    // IM5K4-PPM: 1 Axis
    {attribute 'pytmc' := 'pv: IM5K4:PPM:MMS'}
    {attribute 'TcLinkTo' := '.bLimitForwardEnable  := TIIB[IM5K4-EL7041-E1]^STM Status^Status^Digital input 1;
                              .bLimitBackwardEnable := TIIB[IM5K4-EL7041-E1]^STM Status^Status^Digital input 2;
                              .bBrakeRelease        := TIIB[IM5K4-EL2004-E3]^Channel 1^Output;
                              .nRawEncoderULINT     := TIIB[IM5K4-EL5042-E2]^FB Inputs Channel 1^Position'}
    M17: ST_MotionStage := (sName := 'IM5K4:PPM:MMS');

    // PF1K4-WFS_TARGET: 2 Axes
    {attribute 'pytmc' := 'pv: PF1K4:WFS:MMS:Y'}
    {attribute 'TcLinkTo' := '.bLimitForwardEnable  := TIIB[PF1K4-EL7041-E1]^STM Status^Status^Digital input 1;
                              .bLimitBackwardEnable := TIIB[PF1K4-EL7041-E1]^STM Status^Status^Digital input 2;
                              .bBrakeRelease        := TIIB[PF1K4-EL2004-E4]^Channel 1^Output;
                              .nRawEncoderULINT     := TIIB[PF1K4-EL5042-E3]^FB Inputs Channel 2^Position'}
    M18: ST_MotionStage := (sName := 'PF1K4:WFS:MMS:Y');
    {attribute 'pytmc' := 'pv: PF1K4:WFS:MMS:Z'}
    {attribute 'TcLinkTo' := '.nRawEncoderULINT     := TIIB[PF1K4-EL5042-E3]^FB Inputs Channel 1^Position'}
    M19: ST_MotionStage := (sName := 'PF1K4:WFS:MMS:Z');

    // LI1K4-IP1: 1 Axis
    {attribute 'pytmc' := 'pv: LI1K4:IP1:MMS'}
    {attribute 'TcLinkTo' := '.bLimitForwardEnable  := TIIB[LI1K4-EL7041-E1]^STM Status^Status^Digital input 1;
                              .bLimitBackwardEnable := TIIB[LI1K4-EL7041-E1]^STM Status^Status^Digital input 2;
                              .bBrakeRelease        := TIIB[LI1K4-EL2004-E3]^Channel 1^Output;
                              .nRawEncoderULINT     := TIIB[LI1K4-EL5042-E2]^FB Inputs Channel 1^Position'}
    M20: ST_MotionStage := (sName := 'LI1K4:IP1:MMS');

    // TM1K4: 2 Axes
    {attribute 'pytmc' := 'pv: TM1K4:ATM:MMS:Y'}
    {attribute 'TcLinkTo' := '.bLimitForwardEnable  := TIIB[TM1K4-EL7041-E1]^STM Status^Status^Digital input 1;
                              .bLimitBackwardEnable := TIIB[TM1K4-EL7041-E1]^STM Status^Status^Digital input 2;
                              .bBrakeRelease        := TIIB[TM1K4-EL2004-E4]^Channel 1^Output;
                              .nRawEncoderULINT     := TIIB[TM1K4-EL5042-E3]^FB Inputs Channel 1^Position'}
    M21: ST_MotionStage := (sName := 'TM1K4:ATM:MMS:Y');
    {attribute 'pytmc' := 'pv: TM1K4:ATM:MMS:X'}
    {attribute 'TcLinkTo' := '.nRawEncoderULINT     := TIIB[TM1K4-EL5042-E3]^FB Inputs Channel 2^Position'}
    M22: ST_MotionStage := (sName := 'TM1K4:ATM:MMS:X');

  (*   // SL2K4-SCATTER: 4 Axes
    {attribute 'pytmc' := 'pv: SL2K4:SCATTER:MMS:BOTTOM'}
    {attribute 'TcLinkTo' := '.bLimitForwardEnable  := TIIB[SL2K4-EL7031-E1]^STM Status^Status^Digital input 2;
                             .bLimitBackwardEnable := TIIB[SL2K4-EL7031-E1]^STM Status^Status^Digital input 1;
                              .nRawEncoderUINT      := TIIB[SL2K4-EL5101-E2]^ENC Status compact^Counter value'}
    M23: ST_MotionStage := (sName := 'SL2K4:SCATTER:MMS:BOTTOM');
    {attribute 'pytmc' := 'pv: SL2K4:SCATTER:MMS:TOP'}
    {attribute 'TcLinkTo' := '.bLimitForwardEnable  := TIIB[SL2K4-EL7031-E3]^STM Status^Status^Digital input 2;
                              .bLimitBackwardEnable := TIIB[SL2K4-EL7031-E3]^STM Status^Status^Digital input 1;
                              .nRawEncoderUINT      := TIIB[SL2K4-EL5101-E4]^ENC Status compact^Counter value'}
    M24: ST_MotionStage := (sName := 'SL2K4:SCATTER:MMS:TOP');
    {attribute 'pytmc' := 'pv: SL2K4:SCATTER:MMS:NORTH'}
    {attribute 'TcLinkTo' := '.bLimitForwardEnable  := TIIB[SL2K4-EL7031-E5]^STM Status^Status^Digital input 1;
                              .bLimitBackwardEnable := TIIB[SL2K4-EL7031-E5]^STM Status^Status^Digital input 2;
                              .nRawEncoderUINT      := TIIB[SL2K4-EL5101-E6]^ENC Status compact^Counter value'}
    M25: ST_MotionStage := (sName := 'SL2K4:SCATTER:MMS:NORTH');
    {attribute 'pytmc' := 'pv: SL2K4:SCATTER:MMS:SOUTH'}
    {attribute 'TcLinkTo' := '.bLimitForwardEnable  := TIIB[SL2K4-EL7031-E7]^STM Status^Status^Digital input 1;
                              .bLimitBackwardEnable := TIIB[SL2K4-EL7031-E7]^STM Status^Status^Digital input 2;
                              .nRawEncoderUINT      := TIIB[SL2K4-EL5101-E8]^ENC Status compact^Counter value'}
    M26: ST_MotionStage := (sName := 'SL2K4:SCATTER:MMS:SOUTH');
    *)

    // IM6K4-PPM: 1 Axis
    {attribute 'pytmc' := 'pv: IM6K4:PPM:MMS'}
    {attribute 'TcLinkTo' := '.bLimitForwardEnable  := TIIB[IM6K4-EL7041-E1]^STM Status^Status^Digital input 1;
                              .bLimitBackwardEnable := TIIB[IM6K4-EL7041-E1]^STM Status^Status^Digital input 2;
                              .bBrakeRelease        := TIIB[IM6K4-EL2004-E3]^Channel 1^Output;
                              .nRawEncoderULINT     := TIIB[IM6K4-EL5042-E2]^FB Inputs Channel 1^Position'}
    M27: ST_MotionStage := (sName := 'IM6K4:PPM:MMS');

    // PF2K4-WFS_TARGET: 2 Axes
    {attribute 'pytmc' := 'pv: PF2K4:WFS:MMS:Y'}
    {attribute 'TcLinkTo' := '.bLimitForwardEnable  := TIIB[PF2K4-EL7041-E1]^STM Status^Status^Digital input 1;
                              .bLimitBackwardEnable := TIIB[PF2K4-EL7041-E1]^STM Status^Status^Digital input 2;
                              .bBrakeRelease        := TIIB[PF2K4-EL2004-E4]^Channel 1^Output;
                              .nRawEncoderULINT     := TIIB[PF2K4-EL5042-E3]^FB Inputs Channel 2^Position'}
    M28: ST_MotionStage := (sName := 'PF2K4:WFS:MMS:Y');
    {attribute 'pytmc' := 'pv: PF2K4:WFS:MMS:Z'}
    {attribute 'TcLinkTo' := '.nRawEncoderULINT     := TIIB[PF2K4-EL5042-E3]^FB Inputs Channel 1^Position'}
    M29: ST_MotionStage := (sName := 'PF2K4:WFS:MMS:Z');

    // TM2K4 2 Axes
    {attribute 'pytmc' := 'pv: TM2K4:ATM:MMS:Y'}
    {attribute 'TcLinkTo' := '.bLimitForwardEnable  := TIIB[TM2K4-EL7041-E1]^STM Status^Status^Digital input 1;
                              .bLimitBackwardEnable := TIIB[TM2K4-EL7041-E1]^STM Status^Status^Digital input 2;
                              .bBrakeRelease        := TIIB[TM2K4-EL2004-E4]^Channel 1^Output;
                              .nRawEncoderULINT     := TIIB[TM2K4-EL5042-E3]^FB Inputs Channel 1^Position'}
    M30: ST_MotionStage := (sName := 'TM2K4:ATM:MMS:Y');
    {attribute 'pytmc' := 'pv: TM2K4:ATM:MMS:X'}
    {attribute 'TcLinkTo' := '.nRawEncoderULINT     := TIIB[TM2K4-EL5042-E3]^FB Inputs Channel 2^Position'}
    M31: ST_MotionStage := (sName := 'TM2K4:ATM:MMS:X');

    // SP1K4 14 Axes
    {attribute 'pytmc' := '
        pv: TMO:SPEC:MMS:01
    '}
    // Lens X (not use it after July 2023)
    M32 : ST_MotionStage := (
        bHardwareEnable:=TRUE,
        bPowerSelf:=TRUE,
        nEnableMode:=ENUM_StageEnableMode.DURING_MOTION,
        nHomingMode := ENUM_EpicsHomeCmd.ABSOLUTE_SET);
    {attribute 'TcLinkTo' := '.bLimitForwardEnable:=TIIB[FoilX-EL7041]^STM Status^Status^Digital input 2;
                              .bLimitBackwardEnable:=TIIB[FoilX-EL7041]^STM Status^Status^Digital input 1'
                              .nRawEncoderULINT:=TIIB[SP1K4-EL5042-E2]^FB Inputs Channel 2^Position'}
    {attribute 'pytmc' := '
        pv: TMO:SPEC:MMS:02
    '}
    // solid atten X(Foil X)
    M33: ST_MotionStage := (
        bHardwareEnable:=TRUE,
        bPowerSelf:=FALSE,
        nEnableMode:=ENUM_StageEnableMode.DURING_MOTION,
        nHomingMode := ENUM_EpicsHomeCmd.NONE,
        sName := 'TMO:SPEC:MMS:02');
    {attribute 'TcLinkTo' := '.bLimitForwardEnable:=TIIB[ZonePlateX-EL7041]^STM Status^Status^Digital input 2;
                              .bLimitBackwardEnable:=TIIB[ZonePlateX-EL7041]^STM Status^Status^Digital input 1'
                              .nRawEncoderULINT:=TIIB[SP1K4-EL5042-E1]^FB Inputs Channel 1^Position'}
    {attribute 'pytmc' := '
        pv: TMO:SPEC:MMS:03
    '}
    // Zone Plate X
    M34 : ST_MotionStage := (
        bHardwareEnable:=TRUE,
        bPowerSelf:=FALSE,
        nEnableMode:=ENUM_StageEnableMode.DURING_MOTION,
        sName := 'TMO:SPEC:MMS:03');
    {attribute 'TcLinkTo' := '.bLimitForwardEnable:=TIIB[ZonePlateY-EL7041]^STM Status^Status^Digital input 2;
                              .bLimitBackwardEnable:=TIIB[ZonePlateY-EL7041]^STM Status^Status^Digital input 1';
                              .nRawEncoderULINT:=TIIB[SP1K4-EL5042-E1]^FB Inputs Channel 2^Position'}
    {attribute 'pytmc' := '
        pv: TMO:SPEC:MMS:04
    '}
    // Zone Plate Y
    M35 : ST_MotionStage := (
        bHardwareEnable:=TRUE,
        bPowerSelf:=FALSE,
        nEnableMode:=ENUM_StageEnableMode.DURING_MOTION,
        sName := 'TMO:SPEC:MMS:04');
    {attribute 'TcLinkTo' := '.bLimitForwardEnable:=TIIB[ZonePlateZ-EL7041]^STM Status^Status^Digital input 1;
                              .bLimitBackwardEnable:=TIIB[ZonePlateZ-EL7041]^STM Status^Status^Digital input 2';
                              .nRawEncoderULINT:=TIIB[SP1K4-EL5042-E2]^FB Inputs Channel 1^Position'}
    {attribute 'pytmc' := '
        pv: TMO:SPEC:MMS:05
    '}
    // Zone Plate Z
    M36 : ST_MotionStage := (
        bHardwareEnable:=TRUE,
        bPowerSelf:=FALSE,
        nEnableMode:=ENUM_StageEnableMode.DURING_MOTION,
        sName := 'TMO:SPEC:MMS:05');
    {attribute 'TcLinkTo' := '.bLimitForwardEnable:=TIIB[YagX-EL7041]^STM Status^Status^Digital input 2;
                              .bLimitBackwardEnable:=TIIB[YagX-EL7041]^STM Status^Status^Digital input 1';
                              .nRawEncoderULINT:=TIIB[SP1K4-EL5042-E8]^FB Inputs Channel 1^Position'}

    {attribute 'pytmc' := '
        pv: TMO:SPEC:MMS:06
    '}
    // Yag X
    M37 : ST_MotionStage := (
        bHardwareEnable:=TRUE,
        bPowerSelf:=TRUE,
        nEnableMode:=ENUM_StageEnableMode.DURING_MOTION,
        nHomingMode := ENUM_EpicsHomeCmd.ABSOLUTE_SET);
    {attribute 'TcLinkTo' := '.bLimitForwardEnable:=TIIB[YagY-EL7041]^STM Status^Status^Digital input 1;
                              .bLimitBackwardEnable:=TIIB[YagY-EL7041]^STM Status^Status^Digital input 2'}

    {attribute 'pytmc' := '
        pv: TMO:SPEC:MMS:07
    '}
    // Yag Y
    M38 : ST_MotionStage := (
        bHardwareEnable:=TRUE,
        bPowerSelf:=TRUE,
        nEnableMode:=ENUM_StageEnableMode.DURING_MOTION,
        nHomingMode := ENUM_EpicsHomeCmd.ABSOLUTE_SET);

    {attribute 'TcLinkTo' := '.bLimitForwardEnable:=TIIB[YagZ-EL7041]^STM Status^Status^Digital input 2;
                              .bLimitBackwardEnable:=TIIB[YagZ-EL7041]^STM Status^Status^Digital input 1';
                              .nRawEncoderULINT:=TIIB[SP1K4-EL5042-E8]^FB Inputs Channel 2^Position'}

    {attribute 'pytmc' := '
        pv: TMO:SPEC:MMS:08
    '}
    // Yag Z
    M39 : ST_MotionStage := (
        bHardwareEnable:=TRUE,
        bPowerSelf:=TRUE,
        nEnableMode:=ENUM_StageEnableMode.DURING_MOTION,
        nHomingMode := ENUM_EpicsHomeCmd.ABSOLUTE_SET);
    {attribute 'TcLinkTo' := '.bLimitForwardEnable:=TIIB[YagTheta-EL7041]^STM Status^Status^Digital input 1;
                              .bLimitBackwardEnable:=TIIB[YagTheta-EL7041]^STM Status^Status^Digital input 2'}
    {attribute 'pytmc' := '
        pv: TMO:SPEC:MMS:09
    '}
    // Yag Theta
    M40 : ST_MotionStage := (
        bHardwareEnable:=TRUE,
        bPowerSelf:=TRUE,
        nEnableMode:=ENUM_StageEnableMode.DURING_MOTION,
        nHomingMode := ENUM_EpicsHomeCmd.ABSOLUTE_SET);
    {attribute 'pytmc' := '
        pv: TMO:SPEC:MMS:10
    '}
    // Thorlabs1
    M41 : ST_MotionStage := (
        bHardwareEnable:=TRUE,
        bPowerSelf:=TRUE,
        nEnableMode:=ENUM_StageEnableMode.DURING_MOTION,
        nHomingMode := ENUM_EpicsHomeCmd.ABSOLUTE_SET);
    {attribute 'pytmc' := '
        pv: TMO:SPEC:MMS:11
    '}
    // Thorlabs2
    M42 : ST_MotionStage := (
        bHardwareEnable:=TRUE,
        bPowerSelf:=TRUE,
        nEnableMode:=ENUM_StageEnableMode.DURING_MOTION,
        nHomingMode := ENUM_EpicsHomeCmd.ABSOLUTE_SET);

    {attribute 'pytmc' := '
        pv: TMO:SPEC:MMS:12
    '}
    //thorlab-lenX
    M43 : ST_MotionStage := (
        bHardwareEnable:=TRUE,
        bPowerSelf:=TRUE,
        nEnableMode:=ENUM_StageEnableMode.DURING_MOTION,
        nHomingMode := ENUM_EpicsHomeCmd.ABSOLUTE_SET);

    {attribute 'TcLinkTo' := '.bLimitForwardEnable:=TIIB[FoilY-EL7041]^STM Status^Status^Digital input 1;
                              .bLimitBackwardEnable:=TIIB[FoilY-EL7041]^STM Status^Status^Digital input 2';
                               .nRawEncoderULINT:=TIIB[SP1K4-EL5042-E7]^FB Inputs Channel 2^Position'}
    {attribute 'pytmc' := '
        pv: TMO:SPEC:MMS:13
    '}
     //Solid att Y(FOIL-Y)
    M44 : ST_MotionStage := (
        bHardwareEnable:=TRUE,
        bPowerSelf:=FALSE,
        nEnableMode:=ENUM_StageEnableMode.DURING_MOTION,
        nHomingMode := ENUM_EpicsHomeCmd.NONE,
        sName := 'TMO:SPEC:MMS:13');

 // LI2K4-MMS: Y

    {attribute 'TcLinkTo' := '.bLimitForwardEnable  := TIIB[LI2K4Y-EL7047-E1]^STM Status^Status^Digital input 1;
                              .bLimitBackwardEnable := TIIB[LI2K4Y-EL7047-E1]^STM Status^Status^Digital input 2;
                              .nRawEncoderULINT     := TIIB[LI2K4-EL5042-E2]^FB Inputs Channel 1^Position'}
    {attribute 'pytmc' := '
        pv: LI2K4:IP1:MMS:Y
    '}

    M45: ST_MotionStage := (
        bHardwareEnable:=TRUE,
        bPowerSelf:=FALSE,
        nEnableMode:=ENUM_StageEnableMode.DURING_MOTION,
        nHomingMode := ENUM_EpicsHomeCmd.NONE,
        sName := 'LI2K4:IP1:MMS:Y');
// LI2K4-MMS: X
    {attribute 'TcLinkTo' := '.bLimitForwardEnable  := TIIB[LI2K4X-EL7047-E3]^STM Status^Status^Digital input 1;
                              .bLimitBackwardEnable := TIIB[LI2K4X-EL7047-E3]^STM Status^Status^Digital input 2;
                              .nRawEncoderULINT     := TIIB[LI2K4-EL5042-E2]^FB Inputs Channel 2^Position'}
    {attribute 'pytmc' := '
        pv: LI2K4:IP1:MMS:X
    '}
    M46: ST_MotionStage := (
        bHardwareEnable:=TRUE,
        bPowerSelf:=FALSE,
        nEnableMode:=ENUM_StageEnableMode.DURING_MOTION,
        nHomingMode := ENUM_EpicsHomeCmd.NONE,
        sName := 'LI2K4:IP1:MMS:X');

    //PA1K4-PF-MMS-Y
     {attribute 'TcLinkTo' := '.bLimitForwardEnable  := TIIB[PA1K4-PF-EL7047-E4]^STM Status^Status^Digital input 1;
                              .bLimitBackwardEnable := TIIB[PA1K4-PF-EL7047-E4]^STM Status^Status^Digital input 2;
                              .nRawEncoderULINT     := TIIB[PA1K4-PF-EL5042-E5]^FB Inputs Channel 1^Position'}
    {attribute 'pytmc' := '
        pv: PA1K4:PF:MMS:Y
    '}
    M47: ST_MotionStage := (
        bHardwareEnable:=TRUE,
        bPowerSelf:=FALSE,
        nEnableMode:=ENUM_StageEnableMode.DURING_MOTION,
        nHomingMode := ENUM_EpicsHomeCmd.NONE,
        sName := 'PA1K4:PF:MMS:Y');

END_VAR

// ---- POUs/FB_SP_ZP.TcPOU
FUNCTION_BLOCK FB_SP_ZP
VAR_IN_out
     stXStage: ST_MotionStage;
     stYStage: ST_MotionStage;
     stZStage: ST_MotionStage;
    fbArbiter: FB_Arbiter;
    fbFFHWO: FB_HardwareFFOutput;
END_VAR
VAR_INPUT
    stOut: DUT_PositionState;
    stYag: DUT_PositionState;
    stNe1: DUT_PositionState;
    stNe2: DUT_PositionState;
    stNe3: DUT_PositionState;
    st3w1: DUT_PositionState;
    st3w2: DUT_PositionState;
    stO2: DUT_PositionState;
    stO1: DUT_PositionState;
    stTi1: DUT_PositionState;
    stTi2: DUT_PositionState;
    stN1: DUT_PositionState;
    stN2:DUT_PositionState;
    stC1: DUT_PositionState;
    stC2: DUT_PositionState;
    //nTransitionAssertionID: UDINT;
    //nUnknownAssertionID: UDINT;

          {attribute 'pytmc' := '
        pv: MMS:X:STATE
        io: i
    '}
    fbStates_x: FB_ZonePlate_States;

       {attribute 'pytmc' := '
        pv: MMS:Y:STATE
        io: i
    '}
    fbStates_y: FB_ZonePlate_States;

    zp_enumSet : ENUM_ZonePlate_States;
END_VAR
VAR
     fbXStage: FB_MotionStage;
     fbYStage: FB_MotionStage;
     fbZStage: FB_MotionStage;

    (*FFO*)

    FFO: FB_fastFault :=(
        i_DevName:= 'SP1K4',
        i_Desc := 'Fault Occures when the X and Y states d not match',
        i_TypeCode := 16#300 //todo find a type code on confluence
        );


END_VAR

fbXStage(stMotionStage:=stXStage);
stXStage.bHardwareEnable := TRUE;
stXStage.bPowerSelf := FALSE;
stXStage.nEnableMode := ENUM_StageEnableMode.DURING_MOTION;

fbYStage(stMotionStage:=stYStage);
stYStage.bHardwareEnable := TRUE;
stYStage.bPowerSelf := FALSE;
stYStage.nEnableMode := ENUM_StageEnableMode.DURING_MOTION;

fbZStage(stMotionStage:=stZStage);
stZStage.bHardwareEnable := TRUE;
stZStage.bPowerSelf := FALSE;
stZStage.nEnableMode := ENUM_StageEnableMode.DURING_MOTION;





//TODO write the Y and X position before calling the function

fbStates_X(
    fbArbiter:=fbArbiter,
    fbFFHWO:=fbFFHWO,
 //   nTransitionAssertionID:=nTransitionAssertionID,
 //   nUnknownAssertionID:=nUnknownAssertionID,
    stMotionStage:=stXStage,
    bEnable:=TRUE,
    enumSet:= zp_enumSet,
    stOut:=stOut,
    stYag :=stYag,
    stNe1:=stNe1,
    stNe2:=stNe2,
    stNe3:=stNe3,
    st3w1:=st3w1,
    st3w2:=st3w2,
    stO2:=stO2,
    stO1:=stO1,
    stTi1:=stTi1,
    stTi2:=stTi2,
    stN1:=stN1,
    stN2:=stN2,
    stC1:=stC1,
    stC2:=stC2,
  ); //TODO ADD all other states




fbStates_Y(
    fbArbiter:=fbArbiter,
    fbFFHWO:=fbFFHWO,
 //   nTransitionAssertionID:=nTransitionAssertionID,
//    nUnknownAssertionID:=nUnknownAssertionID,
    stMotionStage:=stYStage,
    bEnable:=TRUE,
    enumSet:= zp_enumSet,
    stOut:=stOut,
    stYag:=stYag,
    stNe1:=stNe1,
    stNe2:=stNe2,
    stNe3:=stNe3,
    st3w1:=st3w1,
    st3w2:=st3w2,
    stO2:=stO2,
    stO1:=stO1,
    stTi1:=stTi1,
    stTi2:=stTi2,
    stN1:=stN1,
    stN2:=stN2,
    stC1:=stC1,
    stC2:=stC2,
);


    FFO(i_xOK:= (fbStates_X.enumGet = fbStates_Y.enumGet),
    io_fbFFHWO:= fbFFHWO,
    i_xAutoReset := TRUE );

END_FUNCTION_BLOCK

// ---- POUs/temp/FB_ZonePlate_States.TcPOU
FUNCTION_BLOCK FB_ZonePlate_States EXTENDS FB_PositionStateBase_WithPMPS
VAR_INPUT
     {attribute 'pytmc' := '
        pv: SET
        io: io
    '}
    enumSet: ENUM_ZonePlate_States;
    stOut: DUT_PositionState;
    stYag: DUT_PositionState;
    stNe1: DUT_PositionState;
    stNe2: DUT_PositionState;
    stNe3: DUT_PositionState;
    st3w1: DUT_PositionState;
    st3w2: DUT_PositionState;
    stO1: DUT_PositionState;
    stO2: DUT_PositionState;
    stTi1: DUT_PositionState;
    stTi2: DUT_PositionState;
    stN1: DUT_PositionState;
    stN2:DUT_PositionState;
    stC1: DUT_PositionState;
    stC2: DUT_PositionState;
    stW1: DuT_PositionState;
END_VAR
VAR_OUTPUT
     {attribute 'pytmc' := '
        pv: GET
        io: i
    '}
    enumGet: ENUM_ZonePlate_States;
END_VAR
VAR
    bInittwo: BOOL := TRUE;
    fbStateDefaults: FB_PositionState_Defaults;
    // These are the default values
    // Set values on states prior to passing in for non-default values
    //TODO correct these default positions
    fDelta: LREAL := 1;
    fVelocity: LREAL := 5;
    fAccel: LREAL := 200;
    fDecel: LREAL := 25;
END_VAR

//State init
IF (bInittwo) THEN
    bInittwo := FALSE;
    //Set theses for every state
    stOut.sName := 'OUT';
    stOut.bUseRawCounts:= FALSE;
    stOut.bValid := TRUE;
        fbStateDefaults(
        stPositionState:=stOut,
        fVeloDefault:=fVelocity,
        fDeltaDefault:=fDelta,
        fAccelDefault:=fAccel,
        fDecelDefault:=fDecel,
    );
    stYag.sName := 'Yag';
    stYag.bUseRawCounts:= FALSE;
    stYag.bValid := TRUE;
        fbStateDefaults(
        stPositionState:=stYag,
        fVeloDefault:=fVelocity,
        fDeltaDefault:=fDelta,
        fAccelDefault:=fAccel,
        fDecelDefault:=fDecel,
    );
    stNe1.sName := 'Ne1';
    stNe1.bUseRawCounts:= FALSE;
    stNe1.bValid := TRUE;
        fbStateDefaults(
        stPositionState:=stNe1,
        fVeloDefault:=fVelocity,
        fDeltaDefault:=fDelta,
        fAccelDefault:=fAccel,
        fDecelDefault:=fDecel,
    );
    stNe2.sName := 'Ne2';
    stNe2.bUseRawCounts:= FALSE;
    stNe2.bValid := TRUE;
        fbStateDefaults(
        stPositionState:=stNe2,
        fVeloDefault:=fVelocity,
        fDeltaDefault:=fDelta,
        fAccelDefault:=fAccel,
        fDecelDefault:=fDecel,
    );
    stNe3.sName := 'Ne3';
    stNe3.bUseRawCounts:= FALSE;
    stNe3.bValid := TRUE;
        fbStateDefaults(
        stPositionState:=stNe3,
        fVeloDefault:=fVelocity,
        fDeltaDefault:=fDelta,
        fAccelDefault:=fAccel,
        fDecelDefault:=fDecel,
    );
    st3w1.sName := '3w1';
    st3w1.bUseRawCounts:= FALSE;
    st3w1.bValid := TRUE;
        fbStateDefaults(
        stPositionState:=st3w1,
        fVeloDefault:=fVelocity,
        fDeltaDefault:=fDelta,
        fAccelDefault:=fAccel,
        fDecelDefault:=fDecel,
    );
    st3w2.sName := '3w2';
    st3w2.bUseRawCounts:= FALSE;
    st3w2.bValid := TRUE;
        fbStateDefaults(
        stPositionState:=st3w2,
        fVeloDefault:=fVelocity,
        fDeltaDefault:=fDelta,
        fAccelDefault:=fAccel,
        fDecelDefault:=fDecel,
    );
    stO1.sName := 'O1';
    stO1.bUseRawCounts:= FALSE;
    stO1.bValid := TRUE;
        fbStateDefaults(
        stPositionState:=stO1,
        fVeloDefault:=fVelocity,
        fDeltaDefault:=fDelta,
        fAccelDefault:=fAccel,
        fDecelDefault:=fDecel,
    );
    stO2.sName := 'O2';
    stO2.bUseRawCounts:= FALSE;
    stO2.bValid := TRUE;
        fbStateDefaults(
        stPositionState:=stO2,
        fVeloDefault:=fVelocity,
        fDeltaDefault:=fDelta,
        fAccelDefault:=fAccel,
        fDecelDefault:=fDecel,
    );

    stTi1.sName := 'Ti1';
    stTi1.bUseRawCounts:= FALSE;
    stTi1.bValid := TRUE;
        fbStateDefaults(
        stPositionState:=stTi1,
        fVeloDefault:=fVelocity,
        fDeltaDefault:=fDelta,
        fAccelDefault:=fAccel,
        fDecelDefault:=fDecel,
    );
    stTi2.sName := 'Ti2';
    stTi2.bUseRawCounts:= FALSE;
    stTi2.bValid := TRUE;
        fbStateDefaults(
        stPositionState:=stTi2,
        fVeloDefault:=fVelocity,
        fDeltaDefault:=fDelta,
        fAccelDefault:=fAccel,
        fDecelDefault:=fDecel,
    );
    stN1.sName := 'N1';
    stN1.bUseRawCounts:= FALSE;
    stN1.bValid := TRUE;
        fbStateDefaults(
        stPositionState:=stN1,
        fVeloDefault:=fVelocity,
        fDeltaDefault:=fDelta,
        fAccelDefault:=fAccel,
        fDecelDefault:=fDecel,
    );
    stN2.sName := 'N2';
    stN2.bUseRawCounts:= FALSE;
    stN2.bValid := TRUE;
        fbStateDefaults(
        stPositionState:=stN2,
        fVeloDefault:=fVelocity,
        fDeltaDefault:=fDelta,
        fAccelDefault:=fAccel,
        fDecelDefault:=fDecel,
    );
    stC1.sName := 'C1';
    stC1.bUseRawCounts:= FALSE;
    stC1.bValid := TRUE;
        fbStateDefaults(
        stPositionState:=stC1,
        fVeloDefault:=fVelocity,
        fDeltaDefault:=fDelta,
        fAccelDefault:=fAccel,
        fDecelDefault:=fDecel,
    );
    stC2.sName := 'C2';
    stC2.bUseRawCounts:= FALSE;
    stC2.bValid := TRUE;
        fbStateDefaults(
        stPositionState:=stC2,
        fVeloDefault:=fVelocity,
        fDeltaDefault:=fDelta,
        fAccelDefault:=fAccel,
        fDecelDefault:=fDecel,
    );
    stW1.sName := 'W1';
    stW1.bUseRawCounts:= FALSE;
    stW1.bValid := TRUE;
        fbStateDefaults(
        stPositionState:=stW1,
        fVeloDefault:=fVelocity,
        fDeltaDefault:=fDelta,
        fAccelDefault:=fAccel,
        fDecelDefault:=fDecel,
    );

//Add all states

    arrStates[1] := stOut;
    arrStates[2] := stYag;
    arrStates[3] := stNe1;
    arrStates[4] := stNe2;
    arrStates[5] := stNe3;
    arrStates[6] := st3w1;
    arrStates[7] := st3w2;
    arrStates[8] := stO1;
    arrStates[9] := stO2;
    arrStates[10] := stTi1;
    arrStates[11] := stTi2;
    arrStates[12] := stN1;
    arrStates[13] := stN2;
    arrStates[14] := stC1;
    arrStates[15] := stC2;
 //   arrStates[16] := stW1;

END_IF

setState := enumSet;
Exec();
enumGet := getState;
enumSet := setState;

END_FUNCTION_BLOCK

// ---- POUs/PRG_1_PlcTask.TcPOU
PROGRAM PRG_1_PlcTask
VAR
END_VAR

PRG_2_PMPS_PRE();

PRG_AL1K4_L2SI();
PRG_IM2K4_PPM();
PRG_IM3K4_PPM();
PRG_IM4K4_PPM();
PRG_IM5K4_PPM();
PRG_IM6K4_PPM();
PRG_LI1K4_IP1();
PRG_PF1K4_WFS_TARGET();
PRG_PF2K4_WFS_TARGET();
PRG_SL1K4_SCATTER();
//PRG_SL2K4_SCATTER();
PRG_ST4K4_TMO_TERM();
PRG_PC5K4();
//PRG_ST5K4_TMO_TERM_FIXED();
PRG_TM1K4();
PRG_TM2K4();
PRG_SP1K4();
PRG_LI2K4_IP1();
PRG_PA1K4_PF();


PRG_3_PMPS_POST();
PRG_4_LOG();

END_PROGRAM

// ---- POUs/PRG_2_PMPS_PRE.TcPOU
PROGRAM PRG_2_PMPS_PRE
VAR
END_VAR

MOTION_GVL.fbStandardPMPSDB(
    io_fbFFHWO:=GVL_PMPS.fbFastFaultOutput1,
    bEnable:=TRUE,
    sPLCName:='plc-tmo-motion',
    sDirectory:='/home/ecs-user/pmpsdb/'
    );

END_PROGRAM

// ---- POUs/PRG_AL1K4_L2SI.TcPOU
PROGRAM PRG_AL1K4_L2SI
VAR
    {attribute 'pytmc' := '
        pv: AL1K4:L2SI
        io: io
    '}
    {attribute 'TcLinkTo' := '.fbLaser.iLaserINT := TIIB[AL1K4-EL4004-E4]^AO Outputs Channel 1^Analog output;
                              .fbLaser.iShutdownINT := TIIB[AL1K4-EL4004-E4]^AO Outputs Channel 2^Analog output'}
    fbAL1K4: FB_REF;
    fbStateSetup: FB_StateSetupHelper;
    stDefault: ST_PositionState :=(
        fVelocity := 1,
        bMoveOK := TRUE,
        bValid := TRUE
    );
//    bInit: BOOL;
END_VAR


fbStateSetup(StPositionState:=stDefault, bSetDefault:=TRUE);
fbStateSetup(StPositionState:=fbAL1K4.stOut, fposition:=-33.5, sPmpsState := 'AL1K4:L2SI-OUT');
fbStateSetup(StPositionState:=fbAL1K4.stIn, fposition:=-75, sPmpsState := 'AL1K4:L2SI-IN');
{*
//fbAL1K4.stOut.fPosition := -33.5; // Upper limit
fbAL1K4.stOut.bUseRawCounts := FALSE;
fbAL1K4.stOut.bValid := TRUE;
fbAL1K4.stOut.bMoveOk := TRUE;
fbAL1K4.stOut.stPMPS.sPmpsState := 'AL1K4:L2SI-OUT';

//fbAL1K4.stIn.fPosition := -75; // Current position at time of edit
fbAL1K4.stIn.bUseRawCounts := FALSE;
fbAL1K4.stIn.bValid := TRUE;
fbAL1K4.stIn.bMoveOk := TRUE;
fbAL1K4.stIn.stPMPS.sPmpsState := 'AL1K4:L2SI-IN';

IF NOT bInit THEN
   bInit := TRUE;
   fbAL1K4.stOut.fPosition := -33.5;
   fbAL1K4.stIn.fPosition := -75;
END_IF
*}
fbAL1K4(
    stYStage := Main.M1,
    fbArbiter := fbArbiter,
    fbFFHWO := fbFastFaultOutput1,
    sDeviceName := 'AL1K4:L2SI',
    sTransitionKey := 'AL1K4:L2SI-TRANSITION',
    bEnableMotion := TRUE,
    bEnableBeamParams := TRUE,
    bEnablePositionLimits := TRUE,
);

END_PROGRAM

// ---- POUs/PRG_IM2K4_PPM.TcPOU
PROGRAM PRG_IM2K4_PPM
VAR
    {attribute 'pytmc' := '
        pv: IM2K4:PPM
        io: io
    '}
    {attribute 'TcLinkTo' := '.fbGige.iIlluminatorINT := TIIB[IM2K4-EL4004-E7]^AO Outputs Channel 1^Analog output;
                              .fbGige.bGigePower := TIIB[IM2K4-EL2004-E3]^Channel 2^Output;
                              .fbPowerMeter.iVoltageINT := TIIB[IM2K4-EL3062-E6]^AI Standard Channel 1^Value;
                              .fbPowerMeter.fbTempSensor.bError := TIIB[IM2K4-EL3314-E4]^TC Inputs Channel 1^Status^Error;
                              .fbPowerMeter.fbTempSensor.bUnderrange := TIIB[IM2K4-EL3314-E4]^TC Inputs Channel 1^Status^Underrange;
                              .fbPowerMeter.fbTempSensor.bOverrange := TIIB[IM2K4-EL3314-E4]^TC Inputs Channel 1^Status^Overrange;
                              .fbPowerMeter.fbTempSensor.iRaw := TIIB[IM2K4-EL3314-E4]^TC Inputs Channel 1^Value;
                              .fbYagTempSensor.bError := TIIB[IM2K4-EL3314-E4]^TC Inputs Channel 2^Status^Error;
                              .fbYagTempSensor.bUnderrange := TIIB[IM2K4-EL3314-E4]^TC Inputs Channel 2^Status^Underrange;
                              .fbYagTempSensor.bOverrange := TIIB[IM2K4-EL3314-E4]^TC Inputs Channel 2^Status^Overrange;
                              .fbYagTempSensor.iRaw := TIIB[IM2K4-EL3314-E4]^TC Inputs Channel 2^Value;
                              .fbFlowSwitch.bFlowOk := TIIB[IM2K4-EL1004-E8]^Channel 1^Input'}
    fbIM2K4: FB_PPM;
//    fStartupVelo: LREAL := 13;
    fbStateSetup: FB_StateSetupHelper;
    stDefault: ST_PositionState :=(
        fVelocity := 13,
        bMoveOK := TRUE,
        bValid := TRUE
    );
//    bInit: BOOL;
END_VAR

fbStateSetup(StPositionState:=stDefault, bSetDefault:=TRUE);

fbStateSetup(StPositionState:=fbIM2K4.stOut, fposition:=-8.59, sPmpsState := 'IM2K4:PPM-OUT');
fbStateSetup(StPositionState:=fbIM2K4.stPower, fposition:=-47.69, sPmpsState := 'IM2K4:PPM-POWERMETER');
fbStateSetup(StPositionState:=fbIM2K4.stYag1, fposition:=-71.69, sPmpsState := 'IM2K4:PPM-YAG1');
fbStateSetup(StPositionState:=fbIM2K4.stYag2, fposition:=-97.70, sPmpsState := 'IM2K4:PPM-YAG2');


{*
//fbIM2K4.stOut.fPosition := -8.59;
fbIM2K4.stOut.fVelocity := fStartupVelo;
fbIM2K4.stOut.bUseRawCounts := FALSE;
fbIM2K4.stOut.bValid := TRUE;
fbIM2K4.stOut.bMoveOk := TRUE;
fbIM2K4.stOut.stPMPS.sPmpsState := 'IM2K4:PPM-OUT';

//fbIM2K4.stPower.fPosition := -47.69;
fbIM2K4.stPower.fVelocity := fStartupVelo;
fbIM2K4.stPower.bUseRawCounts := FALSE;
fbIM2K4.stPower.bValid := TRUE;
fbIM2K4.stPower.bMoveOk := TRUE;
fbIM2K4.stPower.stPMPS.sPmpsState := 'IM2K4:PPM-POWERMETER';

//fbIM2K4.stYag1.fPosition := -71.69;
fbIM2K4.stYag1.fVelocity := fStartupVelo;
fbIM2K4.stYag1.bUseRawCounts := FALSE;
fbIM2K4.stYag1.bValid := TRUE;
fbIM2K4.stYag1.bMoveOk := TRUE;
fbIM2K4.stYag1.stPMPS.sPmpsState := 'IM2K4:PPM-YAG1';

//fbIM2K4.stYag2.fPosition := -97.70;
fbIM2K4.stYag2.fVelocity := fStartupVelo;
fbIM2K4.stYag2.bUseRawCounts := FALSE;
fbIM2K4.stYag2.bValid := TRUE;
fbIM2K4.stYag2.bMoveOk := TRUE;
fbIM2K4.stYag2.stPMPS.sPmpsState := 'IM2K4:PPM-YAG2';

IF NOT bInit THEN
   bInit := TRUE;
   fbIM2K4.stOut.fPosition := -8.59;
   fbIM2K4.stPower.fPosition := -47.69;
   fbIM2K4.stYag1.fPosition := -71.69;
   fbIM2K4.stYag2.fPosition := -97.70;

END_IF
*}


fbIM2K4(
    fbArbiter := fbArbiter,
    fbFFHWO := fbFastFaultOutput1,
    stYStage := Main.M9,
    sDeviceName := 'IM2K4:PPM',
    sTransitionKey := 'IM2K4:PPM-TRANSITION',
    bEnableMotion := TRUE,
    bEnableBeamParams := TRUE,
    bEnablePositionLimits := TRUE,
    fResponsivity := 0.0712,
);

END_PROGRAM

// ---- POUs/PRG_IM3K4_PPM.TcPOU
PROGRAM PRG_IM3K4_PPM
VAR
    {attribute 'pytmc' := '
        pv: IM3K4:PPM
        io: io
    '}
    {attribute 'TcLinkTo' := '.fbGige.iIlluminatorINT 					:= TIIB[IM3K4-EL4004-E7]^AO Outputs Channel 1^Analog output;
                              .fbGige.bGigePower 						:= TIIB[IM3K4-EL2004-E3]^Channel 2^Output;
                              .fbPowerMeter.iVoltageINT 				:= TIIB[IM3K4-EL3062-E6]^AI Standard Channel 1^Value;
                              .fbPowerMeter.fbTempSensor.bError 		:= TIIB[IM3K4-EL3314-E4]^TC Inputs Channel 1^Status^Error;
                              .fbPowerMeter.fbTempSensor.bUnderrange	:= TIIB[IM3K4-EL3314-E4]^TC Inputs Channel 1^Status^Underrange;
                              .fbPowerMeter.fbTempSensor.bOverrange 	:= TIIB[IM3K4-EL3314-E4]^TC Inputs Channel 1^Status^Overrange;
                              .fbPowerMeter.fbTempSensor.iRaw 		:= TIIB[IM3K4-EL3314-E4]^TC Inputs Channel 1^Value;
                              .fbYagTempSensor.bError 				:= TIIB[IM3K4-EL3314-E4]^TC Inputs Channel 2^Status^Error;
                              .fbYagTempSensor.bUnderrange 			:= TIIB[IM3K4-EL3314-E4]^TC Inputs Channel 2^Status^Underrange;
                              .fbYagTempSensor.bOverrange 			:= TIIB[IM3K4-EL3314-E4]^TC Inputs Channel 2^Status^Overrange;
                              .fbYagTempSensor.iRaw 					:= TIIB[IM3K4-EL3314-E4]^TC Inputs Channel 2^Value;
                              .fbFlowMeter.iRaw                         := TIIB[IM4K4-EL3052-E5]^AI Standard Channel 1^Value'} //IM3K4 and IM4K4 share the same flow meter
    fbIM3K4: FB_PPM;
    fbStateSetup: FB_StateSetupHelper;
    stDefault: ST_PositionState :=(
        fVelocity := 12,
        bMoveOK := TRUE,
        bValid := TRUE
    );
 //   fStartupVelo: LREAL := 12;
 //   bInit: BOOL;
END_VAR

fbStateSetup(StPositionState:=stDefault, bSetDefault:=TRUE);

fbStateSetup(StPositionState:=fbIM3K4.stOut, fposition:=-5.82, sPmpsState := 'IM3K4:PPM-OUT');
fbStateSetup(StPositionState:=fbIM3K4.stPower, fposition:=-44.92, sPmpsState := 'IM3K4:PPM-POWERMETER');
fbStateSetup(StPositionState:=fbIM3K4.stYag1, fposition:=-68.92, sPmpsState := 'IM3K4:PPM-YAG1');
fbStateSetup(StPositionState:=fbIM3K4.stYag2, fposition:=-94.93, sPmpsState := 'IM3K4:PPM-YAG2');

{*
//fbIM3K4.stOut.fPosition := -5.82;
fbIM3K4.stOut.fVelocity := fStartupVelo;
fbIM3K4.stOut.bUseRawCounts := FALSE;
fbIM3K4.stOut.bValid := TRUE;
fbIM3K4.stOut.bMoveOk := TRUE;
fbIM3K4.stOut.stPMPS.sPmpsState := 'IM3K4:PPM-OUT';

//fbIM3K4.stPower.fPosition := -44.92;
fbIM3K4.stPower.fVelocity := fStartupVelo;
fbIM3K4.stPower.bUseRawCounts := FALSE;
fbIM3K4.stPower.bValid := TRUE;
fbIM3K4.stPower.bMoveOk := TRUE;
fbIM3K4.stPower.stPMPS.sPmpsState := 'IM3K4:PPM-POWERMETER';

//fbIM3K4.stYag1.fPosition := -68.92;
fbIM3K4.stYag1.fVelocity := fStartupVelo;
fbIM3K4.stYag1.bUseRawCounts := FALSE;
fbIM3K4.stYag1.bValid := TRUE;
fbIM3K4.stYag1.bMoveOk := TRUE;
fbIM3K4.stYag1.stPMPS.sPmpsState := 'IM3K4:PPM-YAG1';

//fbIM3K4.stYag2.fPosition := -94.93;
fbIM3K4.stYag2.fVelocity := fStartupVelo;
fbIM3K4.stYag2.bUseRawCounts := FALSE;
fbIM3K4.stYag2.bValid := TRUE;
fbIM3K4.stYag2.bMoveOk := TRUE;
fbIM3K4.stYag2.stPMPS.sPmpsState := 'IM3K4:PPM-YAG2';

IF NOT bInit THEN
   bInit := TRUE;
   fbIM3K4.stOut.fPosition := -5.82;
   fbIM3K4.stPower.fPosition := -44.92;
   fbIM3K4.stYag1.fPosition := -68.92;
   fbIM3K4.stYag2.fPosition := -94.93;
END_IF
*}
fbIM3K4(
    fbArbiter := fbArbiter,
    fbFFHWO := fbFastFaultOutput1,
    stYStage := Main.M15,
    sDeviceName := 'IM3K4:PPM',
    sTransitionKey := 'IM3K4:PPM-TRANSITION',
    bEnableMotion := TRUE,
    bEnableBeamParams := TRUE,
    bEnablePositionLimits := TRUE,
    fFlowOffset := 0.0,
    fResponsivity := 0.0751,
);

END_PROGRAM

// ---- POUs/PRG_IM4K4_PPM.TcPOU
PROGRAM PRG_IM4K4_PPM
VAR
    {attribute 'pytmc' := '
        pv: IM4K4:PPM
        io: io
    '}
    {attribute 'TcLinkTo' := '.fbGige.iIlluminatorINT 					:= TIIB[IM4K4-EL4004-E7]^AO Outputs Channel 1^Analog output;
                              .fbGige.bGigePower 						:= TIIB[IM4K4-EL2004-E3]^Channel 2^Output;
                              .fbPowerMeter.iVoltageINT 				:= TIIB[IM4K4-EL3062-E6]^AI Standard Channel 1^Value;
                              .fbPowerMeter.fbTempSensor.bError 		:= TIIB[IM4K4-EL3314-E4]^TC Inputs Channel 1^Status^Error;
                              .fbPowerMeter.fbTempSensor.bUnderrange	:= TIIB[IM4K4-EL3314-E4]^TC Inputs Channel 1^Status^Underrange;
                              .fbPowerMeter.fbTempSensor.bOverrange 	:= TIIB[IM4K4-EL3314-E4]^TC Inputs Channel 1^Status^Overrange;
                              .fbPowerMeter.fbTempSensor.iRaw 		:= TIIB[IM4K4-EL3314-E4]^TC Inputs Channel 1^Value;
                              .fbYagTempSensor.bError 				:= TIIB[IM4K4-EL3314-E4]^TC Inputs Channel 2^Status^Error;
                              .fbYagTempSensor.bUnderrange 			:= TIIB[IM4K4-EL3314-E4]^TC Inputs Channel 2^Status^Underrange;
                              .fbYagTempSensor.bOverrange 			:= TIIB[IM4K4-EL3314-E4]^TC Inputs Channel 2^Status^Overrange;
                              .fbYagTempSensor.iRaw 					:= TIIB[IM4K4-EL3314-E4]^TC Inputs Channel 2^Value;
                              .fbFlowMeter.iRaw                         := TIIB[IM4K4-EL3052-E5]^AI Standard Channel 1^Value'}
    fbIM4K4: FB_PPM;
    fbStateSetup: FB_StateSetupHelper;
    stDefault: ST_PositionState :=(
        fVelocity := 15,
        bMoveOK := TRUE,
        bValid := TRUE
    );
//    fStartupVelo: LREAL := 15;
//    bInit: BOOL;
END_VAR

fbStateSetup(StPositionState:=stDefault, bSetDefault:=TRUE);

fbStateSetup(StPositionState:=fbIM4K4.stOut, fposition:=-9.29, sPmpsState := 'IM4K4:PPM-OUT');
fbStateSetup(StPositionState:=fbIM4K4.stPower, fposition:=-48.39, sPmpsState := 'IM4K4:PPM-POWERMETER');
fbStateSetup(StPositionState:=fbIM4K4.stYag1, fposition:=-72.39, sPmpsState := 'IM4K4:PPM-YAG1');
fbStateSetup(StPositionState:=fbIM4K4.stYag2, fposition:=-98.4, sPmpsState := 'IM4K4:PPM-YAG2');

{* //fbIM4K4.stOut.fPosition := -9.29;
fbIM4K4.stOut.fVelocity := fStartupVelo;
fbIM4K4.stOut.bUseRawCounts := FALSE;
fbIM4K4.stOut.bValid := TRUE;
fbIM4K4.stOut.bMoveOk := TRUE;
fbIM4K4.stOut.stPMPS.sPmpsState := 'IM4K4:PPM-OUT';

//fbIM4K4.stPower.fPosition := -48.39;
fbIM4K4.stPower.fVelocity := fStartupVelo;
fbIM4K4.stPower.bUseRawCounts := FALSE;
fbIM4K4.stPower.bValid := TRUE;
fbIM4K4.stPower.bMoveOk := TRUE;
fbIM4K4.stPower.stPMPS.sPmpsState := 'IM4K4:PPM-POWERMETER';

//fbIM4K4.stYag1.fPosition := -72.39;
fbIM4K4.stYag1.fVelocity := fStartupVelo;
fbIM4K4.stYag1.bUseRawCounts := FALSE;
fbIM4K4.stYag1.bValid := TRUE;
fbIM4K4.stYag1.bMoveOk := TRUE;
fbIM4K4.stYag1.stPMPS.sPmpsState := 'IM4K4:PPM-YAG1';

//fbIM4K4.stYag2.fPosition := -98.4;
fbIM4K4.stYag2.fVelocity := fStartupVelo;
fbIM4K4.stYag2.bUseRawCounts := FALSE;
fbIM4K4.stYag2.bValid := TRUE;
fbIM4K4.stYag2.bMoveOk := TRUE;
fbIM4K4.stYag2.stPMPS.sPmpsState := 'IM4K4:PPM-YAG2';

IF Main.M16.fVelocity > 1 AND Main.M16.fVelocity <> 15 AND Main.M16.bExecute THEN
    Main.M16.bError := TRUE;
    Main.M16.nErrorId := 16#4221;
    Main.M16.sCustomErrorMessage := 'Unsafe velocity, try 1 or 15.';
END_IF

IF NOT bInit THEN
   bInit := TRUE;
   fbIM4K4.stOut.fPosition := -9.29;
   fbIM4K4.stPower.fPosition := -48.39;
   fbIM4K4.stYag1.fPosition := -72.39;
   fbIM4K4.stYag2.fPosition := -98.4;
END_IF
*}


fbIM4K4(
    fbArbiter := fbArbiter,
    fbFFHWO := fbFastFaultOutput1,
    stYStage := Main.M16,
    sDeviceName := 'IM4K4:PPM',
    sTransitionKey := 'IM4K4:PPM-TRANSITION',
    bEnableMotion := TRUE,
    bEnableBeamParams := TRUE,
    bEnablePositionLimits := TRUE,
    fFlowOffset := 0.0,
    fResponsivity := 0.0721,
);

END_PROGRAM

// ---- POUs/PRG_IM5K4_PPM.TcPOU
PROGRAM PRG_IM5K4_PPM
VAR
    {attribute 'pytmc' := '
        pv: IM5K4:PPM
        io: io
    '}
    {attribute 'TcLinkTo' := '.fbGige.iIlluminatorINT 					:= TIIB[IM5K4-EL4004-E7]^AO Outputs Channel 1^Analog output;
                              .fbGige.bGigePower 						:= TIIB[IM5K4-EL2004-E3]^Channel 2^Output;
                              .fbPowerMeter.iVoltageINT 				:= TIIB[IM5K4-EL3062-E6]^AI Standard Channel 1^Value;
                              .fbPowerMeter.fbTempSensor.bError 		:= TIIB[IM5K4-EL3314-E4]^TC Inputs Channel 1^Status^Error;
                              .fbPowerMeter.fbTempSensor.bUnderrange	:= TIIB[IM5K4-EL3314-E4]^TC Inputs Channel 1^Status^Underrange;
                              .fbPowerMeter.fbTempSensor.bOverrange 	:= TIIB[IM5K4-EL3314-E4]^TC Inputs Channel 1^Status^Overrange;
                              .fbPowerMeter.fbTempSensor.iRaw 		:= TIIB[IM5K4-EL3314-E4]^TC Inputs Channel 1^Value;
                              .fbYagTempSensor.bError 				:= TIIB[IM5K4-EL3314-E4]^TC Inputs Channel 2^Status^Error;
                              .fbYagTempSensor.bUnderrange 			:= TIIB[IM5K4-EL3314-E4]^TC Inputs Channel 2^Status^Underrange;
                              .fbYagTempSensor.bOverrange 			:= TIIB[IM5K4-EL3314-E4]^TC Inputs Channel 2^Status^Overrange;
                              .fbYagTempSensor.iRaw 					:= TIIB[IM5K4-EL3314-E4]^TC Inputs Channel 2^Value;
                              .fbFlowMeter.iRaw                         := TIIB[IM5K4-EL3052-E5]^AI Standard Channel 1^Value'}
    fbIM5K4: FB_PPM;
    fbStateSetup: FB_StateSetupHelper;
    stDefault: ST_PositionState :=(
        fVelocity := 12,
        bMoveOK := TRUE,
        bValid := TRUE
    );
//    fStartupVelo: LREAL := 12;
   // bInit: BOOL;
END_VAR

fbStateSetup(StPositionState:=stDefault, bSetDefault:=TRUE);

fbStateSetup(StPositionState:=fbIM5K4.stOut, fposition:=-5.13, sPmpsState := 'IM5K4:PPM-OUT');
fbStateSetup(StPositionState:=fbIM5K4.stPower, fposition:=-44.23, sPmpsState := 'IM5K4:PPM-POWERMETER');
fbStateSetup(StPositionState:=fbIM5K4.stYag1, fposition:=-68.23, sPmpsState := 'IM5K4:PPM-YAG1');
fbStateSetup(StPositionState:=fbIM5K4.stYag2, fposition:=-94.24, sPmpsState := 'IM5K4:PPM-YAG2');



//IM5K4 is vetoed by PF1K4
IF( GVL_TcGVL.ePF1K4State >1) THEN//    E_WFS_STATES.TARGET1, E_WFS_STATES.TARGET2, E_WFS_STATES.TARGET3, E_WFS_STATES.TARGET4, E_WFS_STATES.TARGET5 :
        // Known state targets: allow less strict pmps
        fbIM5K4.stYag1.stPMPS.sPmpsState := 'IM5K4:PPM-YAG1_WFS_IN';
        fbIM5K4.stYag2.stPMPS.sPmpsState := 'IM5K4:PPM-YAG2_WFS_IN';

ELSIF (GVL_TcGVL.eSP1K4FZP >1) THEN
        // Known state targets: allow less strict pmps
        fbIM5K4.stYag1.stPMPS.sPmpsState := 'IM5K4:PPM-YAG1_SP1K4_IN';
        fbIM5K4.stYag2.stPMPS.sPmpsState := 'IM5K4:PPM-YAG2_SP1K4_IN';
ELSE
    // Out, Unknown, or an unexpected state: full pmps
    fbIM5K4.stYag1.stPMPS.sPmpsState := 'IM5K4:PPM-YAG1';
    fbIM5K4.stYag2.stPMPS.sPmpsState := 'IM5K4:PPM-YAG2';
END_IF


//IM5K4 is vetoed by SP1K4-FZP
      //paddle1
{*
CASE GVL_TcGVL.eSP1K4FZP OF
    ENUM_ZonePlate_States.FZP290_1, ENUM_ZonePlate_States.FZP290_2, ENUM_ZonePlate_States.FZP410_1, ENUM_ZonePlate_States.FZP410_2, ENUM_ZonePlate_States.FZP460_1, ENUM_ZonePlate_States.FZP460_2, ENUM_ZonePlate_States.FZP530_1,
    ENUM_ZonePlate_States.FZP530_2, ENUM_ZonePlate_States.FZP750_1, ENUM_ZonePlate_States.FZP750_2, ENUM_ZonePlate_States.FZP860_1, ENUM_ZonePlate_States.FZP860_2, ENUM_ZonePlate_States.FZP860_3, ENUM_ZonePlate_States.Yag:
        // Known state targets: allow less strict pmps
        fbIM5K4.stYag1.stPMPS.sPmpsState := 'IM5K4:PPM-YAG1_SP1K4_IN';
        fbIM5K4.stYag2.stPMPS.sPmpsState := 'IM5K4:PPM-YAG2_SP1K4_IN';
ELSE
    // Out, Unknown, or an unexpected state: full pmps
    fbIM5K4.stYag1.stPMPS.sPmpsState := 'IM5K4:PPM-YAG1';
    fbIM5K4.stYag2.stPMPS.sPmpsState := 'IM5K4:PPM-YAG2';
END_CASE
*}

 //paddle2
 (*
CASE GVL_TcGVL.eSP1K4FZP OF
    ENUM_ZonePlate_States.Target1a, ENUM_ZonePlate_States.Target1b, ENUM_ZonePlate_States.Target2a, ENUM_ZonePlate_States.Target2b, ENUM_ZonePlate_States.Target3a, ENUM_ZonePlate_States.Target3b, ENUM_ZonePlate_States.Target4a,
    ENUM_ZonePlate_States.Target4b, ENUM_ZonePlate_States.Target5a, ENUM_ZonePlate_States.Target5b, ENUM_ZonePlate_States.Target6a, ENUM_ZonePlate_States.Target7a, ENUM_ZonePlate_States.Target7b, ENUM_ZonePlate_States.Target6b:
        // Known state targets: allow less strict pmps
        fbIM5K4.stYag1.stPMPS.sPmpsState := 'IM5K4:PPM-YAG1_SP1K4_IN';
        fbIM5K4.stYag2.stPMPS.sPmpsState := 'IM5K4:PPM-YAG2_SP1K4_IN';
ELSE
    // Out, Unknown, or an unexpected state: full pmps
    fbIM5K4.stYag1.stPMPS.sPmpsState := 'IM5K4:PPM-YAG1';
    fbIM5K4.stYag2.stPMPS.sPmpsState := 'IM5K4:PPM-YAG2';
END_CASE
*)

fbIM5K4(
    fbArbiter := fbArbiter,
    fbFFHWO := fbFastFaultOutput1,
    stYStage := Main.M17,
    sDeviceName := 'IM5K4:PPM',
    sTransitionKey := 'IM5K4:PPM-TRANSITION',
    bEnableMotion := TRUE,
    bEnableBeamParams := TRUE,
    bEnablePositionLimits := TRUE,
    fFlowOffset := 0.0,
    fResponsivity := 0.0862,
);

END_PROGRAM

// ---- POUs/PRG_IM6K4_PPM.TcPOU
PROGRAM PRG_IM6K4_PPM
VAR
    {attribute 'pytmc' := '
        pv: IM6K4:PPM
        io: io
    '}
    {attribute 'TcLinkTo' := '.fbGige.iIlluminatorINT 					:= TIIB[IM6K4-EL4004-E7]^AO Outputs Channel 1^Analog output;
                              .fbGige.bGigePower 						:= TIIB[IM6K4-EL2004-E3]^Channel 2^Output;
                              .fbPowerMeter.iVoltageINT 				:= TIIB[IM6K4-EL3062-E6]^AI Standard Channel 1^Value;
                              .fbPowerMeter.fbTempSensor.bError 		:= TIIB[IM6K4-EL3314-E4]^TC Inputs Channel 1^Status^Error;
                              .fbPowerMeter.fbTempSensor.bUnderrange	:= TIIB[IM6K4-EL3314-E4]^TC Inputs Channel 1^Status^Underrange;
                              .fbPowerMeter.fbTempSensor.bOverrange 	:= TIIB[IM6K4-EL3314-E4]^TC Inputs Channel 1^Status^Overrange;
                              .fbPowerMeter.fbTempSensor.iRaw 		:= TIIB[IM6K4-EL3314-E4]^TC Inputs Channel 1^Value;
                              .fbYagTempSensor.bError 				:= TIIB[IM6K4-EL3314-E4]^TC Inputs Channel 2^Status^Error;
                              .fbYagTempSensor.bUnderrange 			:= TIIB[IM6K4-EL3314-E4]^TC Inputs Channel 2^Status^Underrange;
                              .fbYagTempSensor.bOverrange 			:= TIIB[IM6K4-EL3314-E4]^TC Inputs Channel 2^Status^Overrange;
                              .fbYagTempSensor.iRaw 					:= TIIB[IM6K4-EL3314-E4]^TC Inputs Channel 2^Value;
                              .fbFlowMeter.iRaw                         := TIIB[IM6K4-EL3052-E5]^AI Standard Channel 1^Value'}
    fbIM6K4: FB_PPM;
    fbStateSetup: FB_StateSetupHelper;
    stDefault: ST_PositionState :=(
        fVelocity := 13,
        bMoveOK := TRUE,
        bValid := TRUE
    );
//  fStartupVelo: LREAL := 13;
//   bInit: BOOL;
END_VAR

fbStateSetup(StPositionState:=stDefault, bSetDefault:=TRUE);

fbStateSetup(StPositionState:=fbIM6K4.stOut, fposition:=-7.4, sPmpsState := 'IM6K4:PPM-OUT');
fbStateSetup(StPositionState:=fbIM6K4.stPower, fposition:=-46.5, sPmpsState := 'IM6K4:PPM-POWERMETER');
fbStateSetup(StPositionState:=fbIM6K4.stYag1, fposition:=-70.5, sPmpsState := 'IM6K4:PPM-YAG1');
fbStateSetup(StPositionState:=fbIM6K4.stYag2, fposition:=-96.51, sPmpsState := 'IM6K4:PPM-YAG2');

{*//fbIM6K4.stOut.fPosition := -7.4;
fbIM6K4.stOut.fVelocity := fStartupVelo;
fbIM6K4.stOut.bUseRawCounts := FALSE;
fbIM6K4.stOut.bValid := TRUE;
fbIM6K4.stOut.bMoveOk := TRUE;
fbIM6K4.stOut.stPMPS.sPmpsState := 'IM6K4:PPM-OUT';

//fbIM6K4.stPower.fPosition := -46.5;
fbIM6K4.stPower.fVelocity := fStartupVelo;
fbIM6K4.stPower.bUseRawCounts := FALSE;
fbIM6K4.stPower.bValid := TRUE;
fbIM6K4.stPower.bMoveOk := TRUE;
fbIM6K4.stPower.stPMPS.sPmpsState := 'IM6K4:PPM-POWERMETER';

//fbIM6K4.stYag1.fPosition := -70.5;
fbIM6K4.stYag1.fVelocity := fStartupVelo;
fbIM6K4.stYag1.bUseRawCounts := FALSE;
fbIM6K4.stYag1.bValid := TRUE;
fbIM6K4.stYag1.bMoveOk := TRUE;


//fbIM6K4.stYag2.fPosition := -96.51;
fbIM6K4.stYag2.fVelocity := fStartupVelo;
fbIM6K4.stYag2.bUseRawCounts := FALSE;
fbIM6K4.stYag2.bValid := TRUE;
fbIM6K4.stYag2.bMoveOk := TRUE;

*}
CASE GVL_TcGVL.ePF2K4State OF
    E_WFS_STATES.TARGET1, E_WFS_STATES.TARGET2, E_WFS_STATES.TARGET3, E_WFS_STATES.TARGET4, E_WFS_STATES.TARGET5 :
        // Known state targets: allow less strict pmps
        fbIM6K4.stYag1.stPMPS.sPmpsState := 'IM6K4:PPM-YAG1_WFS_IN';
        fbIM6K4.stYag2.stPMPS.sPmpsState := 'IM6K4:PPM-YAG2_WFS_IN';
ELSE
    // Out, Unknown, or an unexpected state: full pmps
    fbIM6K4.stYag1.stPMPS.sPmpsState := 'IM6K4:PPM-YAG1';
    fbIM6K4.stYag2.stPMPS.sPmpsState := 'IM6K4:PPM-YAG2';
END_CASE

{*IF NOT bInit THEN
   bInit := TRUE;
   fbIM6K4.stOut.fPosition := -7.4;
   fbIM6K4.stPower.fPosition := -46.5;
   fbIM6K4.stYag1.fPosition := -70.5;
   fbIM6K4.stYag2.fPosition := -96.51;
END_IF
*}

fbIM6K4(
    fbArbiter := fbArbiter2,
    fbFFHWO := fbFastFaultOutput2,
    stYStage := Main.M27,
    sDeviceName := 'IM6K4:PPM',
    sTransitionKey := 'IM6K4:PPM-TRANSITION',
    bEnableMotion := TRUE,
    bEnableBeamParams := TRUE,
    bEnablePositionLimits := TRUE,
    fFlowOffset := 0.0,
    fResponsivity := 0.0638,
);

END_PROGRAM

// ---- POUs/PRG_LI1K4_IP1.TcPOU
PROGRAM PRG_LI1K4_IP1
VAR
    {attribute 'pytmc' := '
        pv: LI1K4:IP1
        io: io
    '}
    fbLI1K4: FB_LIC;

    fbStateSetup: FB_StateSetupHelper;
    stDefault: ST_PositionState :=(
        fVelocity := 1,
        bMoveOK := TRUE,
        bValid := TRUE
    );
//    stSiBP: ST_BeamParams := PMPS_GVL.cstFullBeam;
//    bInit: BOOL;
END_VAR


// Exclusion range specified by P. Walter 2021-5-19
//stSiBP.neVRange := F_eVExcludeRange(1.6E3, 3.2E3);
// Drop transmission to 20%
//stSiBP.nTran := 0.20;
fbStateSetup(StPositionState:=stDefault, bSetDefault:=TRUE);

fbStateSetup(StPositionState:=fbLI1K4.stOut, fposition:=0.118, sPmpsState := 'LI1K4:IP1-OUT');
fbStateSetup(StPositionState:=fbLI1K4.stMirror1, fposition:=-36.38, sPmpsState := 'LI1K4:IP1-MIRROR1');
fbStateSetup(StPositionState:=fbLI1K4.stMirror2, fposition:=-70.38, sPmpsState := 'LI1K4:IP1-MIRROR2');
fbStateSetup(StPositionState:=fbLI1K4.stTarget1, fposition:=-102.38, sPmpsState := 'LI1K4:IP1-TARGET1');

{* //fbLI1K4.stOut.fPosition := 0.118;
fbLI1K4.stOut.bUseRawCounts := FALSE;
fbLI1K4.stOut.bValid := TRUE;
fbLI1K4.stOut.bMoveOk := TRUE;
fbLI1K4.stOut.stPMPS.sPmpsState := 'LI1K4:IP1-OUT';

//fbLI1K4.stMirror1.fPosition := -36.38;
fbLI1K4.stMirror1.bUseRawCounts := FALSE;
fbLI1K4.stMirror1.bValid := TRUE;
fbLI1K4.stMirror1.bMoveOk := TRUE;
fbLI1K4.stMirror1.stPMPS.sPmpsState := 'LI1K4:IP1-MIRROR1';

//fbLI1K4.stMirror2.fPosition := -70.38;
fbLI1K4.stMirror2.bUseRawCounts := FALSE;
fbLI1K4.stMirror2.bValid := TRUE;
fbLI1K4.stMirror2.bMoveOk := TRUE;
fbLI1K4.stMirror2.stPMPS.sPmpsState := 'LI1K4:IP1-MIRROR2';

//fbLI1K4.stTarget1.fPosition := -102.38;
fbLI1K4.stTarget1.bUseRawCounts := FALSE;
fbLI1K4.stTarget1.bValid := TRUE;
fbLI1K4.stTarget1.bMoveOk := TRUE;
fbLI1K4.stTarget1.stPMPS.sPmpsState := 'LI1K4:IP1-TARGET1';

IF NOT bInit THEN
   bInit := TRUE;
   fbLI1K4.stOut.fPosition := 0.118;
   fbLI1K4.stMirror1.fPosition := -36.38;
   fbLI1K4.stMirror2.fPosition := -70.38;
   fbLI1K4.stTarget1.fPosition := -102.38;
END_IF
*}
fbLI1K4(
    fbArbiter := fbArbiter,
    fbFFHWO := fbFastFaultOutput1,
    stYStage := Main.M20,
    sDeviceName := 'LI1K4:IP1',
    sTransitionKey := 'LI1K4:IP1-TRANSITION',
    bEnableMotion := TRUE,
    bEnableBeamParams := TRUE,
    bEnablePositionLimits := TRUE,
);

END_PROGRAM

// ---- POUs/PRG_PF1K4_WFS_TARGET.TcPOU
  PROGRAM PRG_PF1K4_WFS_TARGET
VAR
    {attribute 'pytmc' := '
        pv: PF1K4:WFS
        io: io
    '}
    {attribute 'TcLinkTo' := '.fbThermoCouple1.bError 		:= TIIB[PF1K4-EL3314-E5]^TC Inputs Channel 1^Status^Error;
                              .fbThermoCouple1.bUnderrange	:= TIIB[PF1K4-EL3314-E5]^TC Inputs Channel 1^Status^Underrange;
                              .fbThermoCouple1.bOverrange 	:= TIIB[PF1K4-EL3314-E5]^TC Inputs Channel 1^Status^Overrange;
                              .fbThermoCouple1.iRaw 		:= TIIB[PF1K4-EL3314-E5]^TC Inputs Channel 1^Value;
                              .fbThermoCouple2.bError 		:= TIIB[PF1K4-EL3314-E5]^TC Inputs Channel 2^Status^Error;
                              .fbThermoCouple2.bUnderrange 	:= TIIB[PF1K4-EL3314-E5]^TC Inputs Channel 2^Status^Underrange;
                              .fbThermoCouple2.bOverrange 	:= TIIB[PF1K4-EL3314-E5]^TC Inputs Channel 2^Status^Overrange;
                              .fbThermoCouple2.iRaw 		:= TIIB[PF1K4-EL3314-E5]^TC Inputs Channel 2^Value;
                              .fbFlowMeter.iRaw             := TIIB[IM5K4-EL3052-E5]^AI Standard Channel 1^Value'} // same cooling loop as IM5K4
    fbPF1K4: FB_WFS;

    fbStateSetup: FB_StateSetupHelper;

    stDefault: ST_PositionState :=(
        fVelocity := 1,
//		bMoveOK := TRUE,
        bValid := TRUE
    );

//    stSiBP: ST_BeamParams := PMPS_GVL.cstFullBeam;

//    bInit: BOOL;
    bSP1K4AttOut: BOOL;
    bSP1K4FzpOut: BOOL;
    bSP1K4Out: BOOL;
END_VAR

bSP1K4AttOut := GVL_TcGVL.eSP1K4ATT = ENUM_SolidAttenuator_States.OUT;
bSP1K4FzpOut := GVL_TcGVL.eSP1K4FZP = ENUM_ZonePlate_States.OUT;
bSP1K4Out := bSP1K4AttOut AND bSP1K4FzpOut;



// Exclusion range specified by M. Seaberg 2021-5-19
//stSiBP.neVRange := F_eVExcludeRange(1.75E3, 3.15E3);
// Drop transmission to 20%
//stSiBP.nTran := 0.20;

fbStateSetup(StPositionState:=stDefault, bSetDefault:=TRUE);

fbStateSetup(StPositionState:=fbPF1K4.stOut, fposition:=-10.5, sPmpsState := 'PF1K4:WFS-OUT');
fbStateSetup(StPositionState:=fbPF1K4.stTarget1, fposition:=-93.033, sPmpsState := 'PF1K4:WFS-TARGET1');
fbStateSetup(StPositionState:=fbPF1K4.stTarget2, fposition:=-78.658, sPmpsState := 'PF1K4:WFS-TARGET2');
fbStateSetup(StPositionState:=fbPF1K4.stTarget3, fposition:=-64.282, sPmpsState := 'PF1K4:WFS-TARGET3');
fbStateSetup(StPositionState:=fbPF1K4.stTarget4, fposition:=-49.907, sPmpsState := 'PF1K4:WFS-TARGET4');
fbStateSetup(StPositionState:=fbPF1K4.stTarget5, fposition:=-35.533, sPmpsState := 'PF1K4:WFS-TARGET5');

fbPF1K4.stOut.bMoveOk := TRUE;
fbPF1K4.stTarget1.bMoveOk := bSP1K4Out;
fbPF1K4.stTarget2.bMoveOk := bSP1K4Out;
fbPF1K4.stTarget3.bMoveOk := bSP1K4Out;
fbPF1K4.stTarget4.bMoveOk := bSP1K4Out;
fbPF1K4.stTarget5.bMoveOk := bSP1K4Out;

{*
//fbPF1K4.stOut.fPosition := -10.5;
fbPF1K4.stOut.bUseRawCounts := FALSE;
fbPF1K4.stOut.bValid := TRUE;
fbPF1K4.stOut.bMoveOk := TRUE;
fbPF1K4.stOut.stPMPS.sPmpsState := 'PF1K4:WFS-OUT';

//fbPF1K4.stTarget1.fPosition := -93.033;
fbPF1K4.stTarget1.bUseRawCounts := FALSE;
fbPF1K4.stTarget1.bValid := TRUE;
fbPF1K4.stTarget1.bMoveOk := TRUE;
fbPF1K4.stTarget1.stPMPS.sPmpsState := 'PF1K4:WFS-TARGET1';

//fbPF1K4.stTarget2.fPosition := -78.658;
fbPF1K4.stTarget2.bUseRawCounts := FALSE;
fbPF1K4.stTarget2.bValid := TRUE;
fbPF1K4.stTarget2.bMoveOk := TRUE;
fbPF1K4.stTarget2.stPMPS.sPmpsState := 'PF1K4:WFS-TARGET2';

//fbPF1K4.stTarget3.fPosition := -64.282;
fbPF1K4.stTarget3.bUseRawCounts := FALSE;
fbPF1K4.stTarget3.bValid := TRUE;
fbPF1K4.stTarget3.bMoveOk := TRUE;
fbPF1K4.stTarget3.stPMPS.sPmpsState := 'PF1K4:WFS-TARGET3';

//fbPF1K4.stTarget4.fPosition := -49.907;
fbPF1K4.stTarget4.bUseRawCounts := FALSE;
fbPF1K4.stTarget4.bValid := TRUE;
fbPF1K4.stTarget4.bMoveOk := TRUE;
fbPF1K4.stTarget4.stPMPS.sPmpsState := 'PF1K4:WFS-TARGET4';

//fbPF1K4.stTarget5.fPosition := -35.533;
fbPF1K4.stTarget5.bUseRawCounts := FALSE;
fbPF1K4.stTarget5.bValid := TRUE;
fbPF1K4.stTarget5.bMoveOk := TRUE;
fbPF1K4.stTarget5.stPMPS.sPmpsState := 'PF1K4:WFS-TARGET5';

 IF NOT bInit THEN
   bInit := TRUE;
   fbPF1K4.stOut.fPosition := -10.5;
   fbPF1K4.stTarget1.fPosition := -93.033;
   fbPF1K4.stTarget2.fPosition := -78.658;
   fbPF1K4.stTarget3.fPosition := -64.282;
   fbPF1K4.stTarget4.fPosition := -49.907;
   fbPF1K4.stTarget5.fPosition := -35.533;

END_IF
*}

fbPF1K4(
    fbArbiter := fbArbiter,
    fbFFHWO := fbFastFaultOutput1,
    stYStage := Main.M18,
    stZStage := Main.M19,
    sDeviceName := 'PF1K4:WFS',
    sTransitionKey := 'PF1K4:WFS-TRANSITION',
    bEnableMotion := TRUE,
    bEnableBeamParams := TRUE,
    bEnablePositionLimits := TRUE,
    eEnumGet => GVL_TcGVL.ePF1K4State,
    );

END_PROGRAM

// ---- POUs/PRG_PF2K4_WFS_TARGET.TcPOU
PROGRAM PRG_PF2K4_WFS_TARGET
VAR
    {attribute 'pytmc' := '
        pv: PF2K4:WFS
        io: io
    '}
    {attribute 'TcLinkTo' := '.fbThermoCouple1.bError 		:= TIIB[PF2K4-EL3314-E5]^TC Inputs Channel 1^Status^Error;
                              .fbThermoCouple1.bUnderrange	:= TIIB[PF2K4-EL3314-E5]^TC Inputs Channel 1^Status^Underrange;
                              .fbThermoCouple1.bOverrange 	:= TIIB[PF2K4-EL3314-E5]^TC Inputs Channel 1^Status^Overrange;
                              .fbThermoCouple1.iRaw 		:= TIIB[PF2K4-EL3314-E5]^TC Inputs Channel 1^Value;
                              .fbThermoCouple2.bError 		:= TIIB[PF2K4-EL3314-E5]^TC Inputs Channel 2^Status^Error;
                              .fbThermoCouple2.bUnderrange 	:= TIIB[PF2K4-EL3314-E5]^TC Inputs Channel 2^Status^Underrange;
                              .fbThermoCouple2.bOverrange 	:= TIIB[PF2K4-EL3314-E5]^TC Inputs Channel 2^Status^Overrange;
                              .fbThermoCouple2.iRaw 		:= TIIB[PF2K4-EL3314-E5]^TC Inputs Channel 2^Value;
                              .fbFlowMeter.iRaw             := TIIB[IM6K4-EL3052-E5]^AI Standard Channel 1^Value'} // same cooling loop as IM6K4
    fbPF2K4: FB_WFS;
    fbStateSetup: FB_StateSetupHelper;
    stDefault: ST_PositionState :=(
        fVelocity := 1,
        bMoveOK := TRUE,
        bValid := TRUE
    );

//    stSiBP: ST_BeamParams := PMPS_GVL.cstFullBeam;
//    bInit: BOOL;
END_VAR

// Exclusion range specified by M. Seaberg 2021-5-19 and James 2022-07-08
//stSiBP.neVRange := F_eVExcludeRange(1.75E3, 3.15E3);
// Drop transmission to 20%
//stSiBP.nTran := 0.20;

fbStateSetup(StPositionState:=stDefault, bSetDefault:=TRUE);

fbStateSetup(StPositionState:=fbPF2K4.stOut, fposition:=-13.5, sPmpsState := 'PF2K4:WFS-OUT');
fbStateSetup(StPositionState:=fbPF2K4.stTarget1, fposition:=-96.127, sPmpsState := 'PF2K4:WFS-TARGET1');
fbStateSetup(StPositionState:=fbPF2K4.stTarget2, fposition:=-81.753, sPmpsState := 'PF2K4:WFS-TARGET2');
fbStateSetup(StPositionState:=fbPF2K4.stTarget3, fposition:=-67.378, sPmpsState := 'PF2K4:WFS-TARGET3');
fbStateSetup(StPositionState:=fbPF2K4.stTarget4, fposition:=-53.002, sPmpsState := 'PF2K4:WFS-TARGET4');
fbStateSetup(StPositionState:=fbPF2K4.stTarget5, fposition:=-38.627, sPmpsState := 'PF2K4:WFS-TARGET5');
{*
//fbPF2K4.stOut.fPosition := -13.5;
fbPF2K4.stOut.bUseRawCounts := FALSE;
fbPF2K4.stOut.bValid := TRUE;
fbPF2K4.stOut.bMoveOk := TRUE;
fbPF2K4.stOut.stPMPS.sPmpsState := 'PF2K4:WFS-OUT';

//fbPF2K4.stTarget1.fPosition := -96.127;
fbPF2K4.stTarget1.bUseRawCounts := FALSE;
fbPF2K4.stTarget1.bValid := TRUE;
fbPF2K4.stTarget1.bMoveOk := TRUE;
fbPF2K4.stTarget1.stPMPS.sPmpsState := 'PF2K4:WFS-TARGET1';

//fbPF2K4.stTarget2.fPosition := -81.753;
fbPF2K4.stTarget2.bUseRawCounts := FALSE;
fbPF2K4.stTarget2.bValid := TRUE;
fbPF2K4.stTarget2.bMoveOk := TRUE;
fbPF2K4.stTarget2.stPMPS.sPmpsState := 'PF2K4:WFS-TARGET2';

//fbPF2K4.stTarget3.fPosition := -67.378;
fbPF2K4.stTarget3.bUseRawCounts := FALSE;
fbPF2K4.stTarget3.bValid := TRUE;
fbPF2K4.stTarget3.bMoveOk := TRUE;
fbPF2K4.stTarget3.stPMPS.sPmpsState := 'PF2K4:WFS-TARGET3';

//fbPF2K4.stTarget4.fPosition := -53.002;
fbPF2K4.stTarget4.bUseRawCounts := FALSE;
fbPF2K4.stTarget4.bValid := TRUE;
fbPF2K4.stTarget4.bMoveOk := TRUE;
fbPF2K4.stTarget4.stPMPS.sPmpsState := 'PF2K4:WFS-TARGET4';

//fbPF2K4.stTarget5.fPosition := -38.627;
fbPF2K4.stTarget5.bUseRawCounts := FALSE;
fbPF2K4.stTarget5.bValid := TRUE;
fbPF2K4.stTarget5.bMoveOk := TRUE;
fbPF2K4.stTarget5.stPMPS.sPmpsState := 'PF2K4:WFS-TARGET5';

IF NOT bInit THEN
   bInit := TRUE;
   fbPF2K4.stOut.fPosition := -13.5;
   fbPF2K4.stTarget1.fPosition := -96.127;
   fbPF2K4.stTarget2.fPosition := -81.753;
   fbPF2K4.stTarget3.fPosition := -67.387;
   fbPF2K4.stTarget4.fPosition := -53.002;
   fbPF2K4.stTarget5.fPosition := -38.627;

END_IF

*}

fbPF2K4(
    fbArbiter := fbArbiter2,
    fbFFHWO := fbFastFaultOutput2,
    stYStage := Main.M28,
    stZStage := Main.M29,
    sDeviceName := 'PF2K4:WFS',
    sTransitionKey := 'PF2K4:WFS-TRANSITION',
    bEnableMotion := TRUE,
    bEnableBeamParams := TRUE,
    bEnablePositionLimits := TRUE,
    eEnumGet => GVL_TcGVL.ePF2K4State,
);

END_PROGRAM

// ---- POUs/PRG_SL1K4_SCATTER.TcPOU
PROGRAM PRG_SL1K4_SCATTER
VAR
    {attribute 'pytmc' := '
        pv: SL1K4:SCATTER
        io: io
    '}
    fbSL1K4: FB_SLITS;
    //GET PMPS Move Ok bit
    // Default True until it is properly linked to PMPS bit
    bMoveOk:BOOL :=TRUE;
    {attribute 'pytmc' := '
    pv: SL1K4:SCATTER:GO;
    io: io;
    field: ZNAM False;
    field: ONAM True;
    '}
    bExecuteMotion :BOOL :=FALSE;
    bTest:BOOL:=FALSE;
    //for testing purposes only. comment-out/delete once done.
    mcPower : ARRAY [1..4] OF MC_POWER;


    (*Offsets*)
    (* Absolute encoder value at the HLS + Absolure eoncoder value at the centered beam *)
    rEncoderOffsetTop: REAL := -15; (* 0+(-15)*)
    rEncoderOffsetBottom: REAL := -15; (* 0+(-15)*)
    rEncoderOffsetNorth: REAL := -15;(* 0+(-15)*)
    rEncoderOffsetSouth: REAL := -15;(* 0+(-15)*)

END_VAR

// M10, Axis 10
// M11, Axis 11
// M12, Axis 12
// M13, Axis 13


fbSL1K4.bMoveOk := bMoveOk;

//for testing purposes only. comment-out/delete once done.
If (bTest) THEN
mcPower[1](axis:=Main.M10.Axis, Enable:=bTest, enable_positive:=Main.M10.bLimitForwardEnable, enable_negative:=Main.M10.bLimitBackwardEnable);
mcPower[2](axis:=Main.M11.Axis, Enable:=bTest, enable_positive:=Main.M11.bLimitForwardEnable, enable_negative:=Main.M11.bLimitBackwardEnable);
mcPower[3](axis:=Main.M12.Axis, Enable:=bTest, enable_positive:=Main.M12.bLimitForwardEnable, enable_negative:=Main.M12.bLimitBackwardEnable);
mcPower[4](axis:=Main.M13.Axis, Enable:=bTest, enable_positive:=Main.M13.bLimitForwardEnable, enable_negative:=Main.M13.bLimitBackwardEnable);
ELSE

//Homing routine parameters
Main.M11.fHomePosition:= 0;
Main.M10.fHomePosition:= -31.5006;
Main.M12.fHomePosition:= 0;
Main.M13.fHomePosition:= -30.23;

Main.M11.nHomingMode := ENUM_EpicsHomeCmd.HIGH_LIMIT;
Main.M10.nHomingMode := ENUM_EpicsHomeCmd.LOW_LIMIT;
Main.M12.nHomingMode := ENUM_EpicsHomeCmd.HIGH_LIMIT;
Main.M13.nHomingMode := ENUM_EpicsHomeCmd.LOW_LIMIT;

fbSL1K4.rEncoderOffsetTop := rEncoderOffsetTop;
fbSL1K4.rEncoderOffsetBottom := rEncoderOffsetBottom;
fbSL1K4.rEncoderOffsetNorth := rEncoderOffsetNorth;
fbSL1K4.rEncoderOffsetSouth := rEncoderOffsetSouth;

fbSL1K4(stTopBlade:=  Main.M11,
        stBottomBlade:= Main.M10,
        stNorthBlade:=  Main.M12,
        stSouthBlade:=  Main.M13,
        bExecuteMotion:=bExecuteMotion,
        io_fbFFHWO := GVL_PMPS.fbFastFaultOutput1,
        fbArbiter := GVL_PMPS.fbArbiter);

fbSL1K4.M_CheckPMPS(2);



//fbSL1K4.M_HomeBlade(stBlade:=Main.M11);
//fbSL1K4.M_HomeBlade(stBlade:=Main.M10);
//fbSL1K4.M_HomeBlade(stBlade:=Main.M12);
//fbSL1K4.M_HomeBlade(stBlade:=Main.M13);

END_IF

END_PROGRAM

// ---- POUs/temp/FB_SLITS.TcPOU
FUNCTION_BLOCK FB_SLITS
VAR_IN_OUT
    stTopBlade: DUT_MotionStage;
    stBottomBlade: DUT_MotionStage;
    stNorthBlade: DUT_MotionStage;
    stSouthBlade: DUT_MotionStage;
    bExecuteMotion:BOOL ;
    io_fbFFHWO    :    FB_HardwareFFOutput;
    fbArbiter: FB_Arbiter();
END_VAR

VAR_INPUT

    {attribute 'pytmc' := '
    pv: PMPS_OK;
    io: i;
    field: ZNAM False
    field: ONAM True
    '}
    bMoveOk:BOOL;

        (*Offsets*)
    {attribute 'pytmc' := '
    pv: Offset_Top;
    io: io;
    '}
    rEncoderOffsetTop: REAL;
    {attribute 'pytmc' := '
    pv: ZeroOffset_Bottom;
    io: io;
    '}
    rEncoderOffsetBottom: REAL;
    {attribute 'pytmc' := '
    pv: ZeroOffset_North;
    io: io;
    '}
    rEncoderOffsetNorth: REAL;
    {attribute 'pytmc' := '
    pv: ZeroOffset_South;
    io: io;
    '}
    rEncoderOffsetSouth: REAL;
    i_DevName : STRING; //device name for FFO and PMPS diagnostics
     {attribute 'pytmc' := '
    pv: Home;
    io: i;
    field: ZNAM False
    field: ONAM True
    '}
    bHome:BOOL:=FALSE;
END_VAR

VAR
    fbTopBlade: FB_MotionStage;
    fbBottomBlade: FB_MotionStage;
    fbNorthBlade: FB_MotionStage;
    fbSouthBlade: FB_MotionStage;
    fPosTopBlade: LREAL;
    fPosBottomBlade: LREAL;
    fPosNorthBlade: LREAL;
    fPosSouthBlade: LREAL;

    (*Motion Parameters*)
    fSmallDelta: LREAL := 0.01;
    fBigDelta: LREAL := 10;
    fMaxVelocity: LREAL := 0.2;
    fHighAccel: LREAL := 0.8;
    fLowAccel: LREAL := 0.1;

    stTop: DUT_PositionState;
    stBOTTOM: DUT_PositionState;
    stNorth: DUT_PositionState;
    stSouth: DUT_PositionState;

    {attribute 'pytmc' := 'pv: TOP'}
    fbTop: FB_StatePTPMove;
    {attribute 'pytmc' := 'pv: BOTTOM'}
    fbBottom: FB_StatePTPMove;
    {attribute 'pytmc' := 'pv: NORTH'}
    fbNorth: FB_StatePTPMove;
    {attribute 'pytmc' := 'pv: SOUTH'}
    fbSouth: FB_StatePTPMove;

    (*EPICS pvs*)
    {attribute 'pytmc' := '
    pv: XWID_REQ;
    io: io;
    '}
    rReqApertureSizeX : REAL;
    {attribute 'pytmc' := '
    pv: YWID_REQ;
    io: io;
    '}
    rReqApertureSizeY : REAL;
    {attribute 'pytmc' := '
    pv: XCEN_REQ;
    io: io;
    '}
    rReqCenterX: REAL;
    {attribute 'pytmc' := '
    pv: YCEN_REQ;
    io: io;
    '}
    rReqCenterY: REAL;

    {attribute 'pytmc' := '
    pv: ACTUAL_XWIDTH;
    io: io;
    '}
    rActApertureSizeX : REAL;

    {attribute 'pytmc' := '
    pv: ACTUAL_YWIDTH;
    io: io;
    '}
    rActApertureSizeY : REAL;
    {attribute 'pytmc' := '
    pv: ACTUAL_XCENTER;
    io: io;
    '}
    rActCenterX: REAL;
    {attribute 'pytmc' := '
    pv: ACTUAL_YCENTER;
    io: io;
    '}
    rActCenterY: REAL;

    {attribute 'pytmc' := '
    pv: XCEN_SETZERO;
    io: io;
    '}
    rSetCenterX: BOOL;
    {attribute 'pytmc' := '
    pv: YCEN_SETZERO;
    io: io;
    '}
    rSetCenterY: BOOL;


    {attribute 'pytmc' := '
    pv: OPEN;
    io: io;
    field: ZNAM False
    field: ONAM True
    '}
    bOpen: BOOL;

    {attribute 'pytmc' := '
    pv: CLOSE;
    io: io;
    field: ZNAM False
    field: ONAM True
    '}
    bClose: BOOL;

    {attribute 'pytmc' := '
    pv: BLOCK;
    io: io;
    field: ZNAM False
    field: ONAM True
    '}
    bBlock: BOOL;


     {attribute 'pytmc' := '
    pv: HOME_READY;
    io: i;
    field: ZNAM False
    field: ONAM True
    '}
    bHomeReady:BOOL:=FALSE;


        //Local variables
    bInit: BOOL :=true;
    rTrig_Block: R_TRIG;
    rTrig_Open: R_TRIG;
    rTrig_Close: R_TRIG;

    //old values
    rOldReqApertureSizeX : REAL;
    rOldReqApertureSizeY : REAL;
    rOldReqCenterX: REAL;
    rOldReqCenterY: REAL;

    bExecuteMotionX: BOOL;
    bExecuteMotionY: BOOL;


    fPosBlock: LREAL;
    fPosClose: LREAL;
    fPosOpen: LREAL;

    stSetPositionOptions:ST_SetPositionOptions;
    fbSetPosition_TOP: MC_SetPosition;
    fbSetPosition_Bottom: MC_SetPosition;
    fbSetPosition_North: MC_SetPosition;
    fbSetPosition_South: MC_SetPosition;

    // For logging
    fbLogger : FB_LogMessage := (eSubsystem:=E_SubSystem.MOTION);
    tErrorPresent : R_TRIG;
    tAction : R_TRIG;
    tOverrideActivated : R_TRIG;

    FFO    :    FB_FastFault :=(
        i_DevName := 'Slits',
        i_Desc := 'Fault occurs when center is greated than that requested',
        i_TypeCode := 16#1010);


    bTest: BOOL;

    AptArrayStatus AT %Q* : ST_PMPS_Aperture_IO;
    AptArrayReq AT %I* : ST_PMPS_Aperture_IO;

END_VAR

ACT_init();

// Instantiate Function block for all the blades
ACT_Motion();
//SET and GET the requested and Actual values
ACT_CalculatePositions();
//ACT_BLOCK();

ACTION ACT_BLOCK:
rTrig_Block (CLK:= bBlock);
rTrig_Open (CLK:= bOpen);
rTrig_Close (CLK:= bClose);

if (rTrig_Block.Q) THEN
    //BLOCK

    bBlock := false;
END_IF

if (rTrig_Open.Q) THEN


    bOpen := false;
END_IF

if (rTrig_Close.Q) THEN


    bClose := false;
END_IF
END_ACTION

ACTION ACT_CalculatePositions:
//check if requested center or gap has changed
//check that the requested values are within acceptable motion range
IF (rOldReqApertureSizeX <> rReqApertureSizeX) THEN
        rOldReqApertureSizeX := rReqApertureSizeX;
        bExecuteMotionX := TRUE;
        fbLogger(sMsg:='Requested new X gap.', eSevr:=TcEventSeverity.Verbose);
END_IF

IF (rOldReqCenterX <> rReqCenterX) THEN
    rOldReqCenterX := rReqCenterX;
    bExecuteMotionX := TRUE;
    fbLogger(sMsg:='Requested new X center', eSevr:=TcEventSeverity.Verbose);
   // ELSE
      //  rReqCenterX := rActCenterX;
END_IF

IF (rOldReqApertureSizeY <> rReqApertureSizeY) THEN
        rOldReqApertureSizeY := rReqApertureSizeY;
        bExecuteMotionY := TRUE;
        fbLogger(sMsg:='Requested new Y gap.', eSevr:=TcEventSeverity.Verbose);

END_IF

IF (rOldReqCenterY <> rReqCenterY) THEN
    rOldReqCenterY := rReqCenterY;
    bExecuteMotionY := TRUE;
    fbLogger(sMsg:='Requested new Y center.', eSevr:=TcEventSeverity.Verbose);
   // ELSE
      //  rReqCenterY := rActCenterY;
END_IF


//Calculate requested target positions from requested gap and center
fPosTopBlade := (rReqApertureSizeY/2) + (rReqCenterY + rEncoderOffsetTop) ;
fPosBottomBlade := (-1*rReqApertureSizeY/2) + (rReqCenterY+rEncoderOffsetBottom);

fPosNorthBlade := (rReqApertureSizeX/2) + (rReqCenterX + rEncoderOffsetNorth);
fPosSouthBlade := (-1*rReqApertureSizeX/2) + (rReqCenterX + rEncoderOffsetSouth);


//Calculate actual gap and center from actual stages positions
rActApertureSizeX := LREAL_TO_REAL((stNorthBlade.stAxisStatus.fActPosition - rEncoderOffsetNorth) - (stSouthBlade.stAxisStatus.fActPosition- rEncoderOffsetSouth));

rActApertureSizeY := LREAL_TO_REAL((stTopBlade.stAxisStatus.fActPosition - rEncoderOffsetTop) - (stBottomBlade.stAxisStatus.fActPosition - rEncoderOffsetBottom));

rActCenterX := LREAL_TO_REAL((((stNorthBlade.stAxisStatus.fActPosition - rEncoderOffsetNorth)  + (stSouthBlade.stAxisStatus.fActPosition - rEncoderOffsetSouth ))/2));

rActCenterY := LREAL_TO_REAL((((stTopBlade.stAxisStatus.fActPosition - rEncoderOffsetTop) + (stBottomBlade.stAxisStatus.fActPosition - rEncoderOffsetBottom))/2));



//Update PMPS Arbiter with the Actual Size and Center of the Aperture
END_ACTION

ACTION ACT_Home:

END_ACTION

ACTION ACT_Init:

//  init the motion stages parameters
IF ( bInit) THEN
    stTopBlade.bHardwareEnable := TRUE;
    stBottomBlade.bHardwareEnable := TRUE;
    stNorthBlade.bHardwareEnable := TRUE;
    stSouthBlade.bHardwareEnable := TRUE;
    stTopBlade.bPowerSelf :=TRUE;
    stBottomBlade.bPowerSelf :=TRUE;
    stNorthBlade.bPowerSelf :=TRUE;
    stSouthBlade.bPowerSelf :=TRUE;
    stTopBlade.nBrakeMode := ENUM_StageBrakeMode.NO_BRAKE;
    stBottomBlade.nBrakeMode := ENUM_StageBrakeMode.NO_BRAKE;
    stNorthBlade.nBrakeMode := ENUM_StageBrakeMode.NO_BRAKE;
    stSouthBlade.nBrakeMode := ENUM_StageBrakeMode.NO_BRAKE;
    FFO.i_DevName := i_DevName;
END_IF
END_ACTION

ACTION ACT_Motion:
// Instantiate Function block for all the blades
fbTopBlade(stMotionStage:=stTopBlade);
fbBottomBlade(stMotionStage:=stBottomBlade);
fbNorthBlade(stMotionStage:=stNorthBlade);
fbSouthBlade(stMotionStage:=stSouthBlade);

// PTP Motion for each blade
stTop.sName := 'Top';
stTop.fPosition := fPosTopBlade;
stTop.fDelta := fSmallDelta;
stTop.fVelocity := fMaxVelocity;
stTop.fAccel := fHighAccel;
stTop.fDecel := fHighAccel;

stBOTTOM.sName := 'Bottom';
stBOTTOM.fPosition := fPosBottomBlade;
stBOTTOM.fDelta := fSmallDelta;
stBOTTOM.fVelocity := fMaxVelocity;
stBOTTOM.fAccel := fHighAccel;
stBOTTOM.fDecel := fHighAccel;

stNorth.sName := 'North';
stNorth.fPosition := fPosNorthBlade;
stNorth.fDelta := fSmallDelta;
stNorth.fVelocity := fMaxVelocity;
stNorth.fAccel := fHighAccel;
stNorth.fDecel := fHighAccel;

stSouth.sName := 'South';
stSouth.fPosition := fPosSouthBlade;
stSouth.fDelta := fSmallDelta;
stSouth.fVelocity := fMaxVelocity;
stSouth.fAccel := fHighAccel;
stSouth.fDecel := fHighAccel;

IF (bExecuteMotionY) THEN
    fbTop.bExecute := fbBottom.bExecute := bExecuteMotionY;
    bExecuteMotionY:= FALSE;
END_IF

IF (bExecuteMotionX) THEN
    fbNorth.bExecute := fbSouth.bExecute := bExecuteMotionX;
    bExecuteMotionX:= FALSE;
END_IF


fbTop(
    stPositionState:=stTop,
    bMoveOk:=bMoveOk,
    stMotionStage:=stTopBlade);

fbBottom(
    stPositionState:=stBOTTOM,
    bMoveOk:=bMoveOk,
    stMotionStage:=stBottomBlade);

fbNorth(
    stPositionState:=stNorth,
    bMoveOk:=bMoveOk,
    stMotionStage:=stNorthBlade);

fbSouth(
    stPositionState:=stSouth,
    bMoveOk:=bMoveOk,
    stMotionStage:=stSouthBlade);
END_ACTION

ACTION ACT_Zero:
//ZERO BIAS

// Set Y center to zero

// Set X center to zero
(*
if (rSetCenterY)THEN
        rSetCenterY := false;
        // Set Current Position
        fbSetPosition_TOP.Position :=  stTopBlade.stAxisStatus.fActPosition - rActCenterY ;
        fbSetPosition_TOP.Execute := TRUE;
        fbSetPosition_Bottom.Position := stBottomBlade.stAxisStatus.fActPosition - rActCenterY;
        fbSetPosition_Bottom.Execute := TRUE;
END_IF

if (rSetCenterX)THEN
        rSetCenterX := false;
        // Set Current Position
        fbSetPosition_North.Position := stNorthBlade.stAxisStatus.fActPosition - rActCenterX ;
        fbSetPosition_North.Execute := TRUE;
        fbSetPosition_South.Position := stSouthBlade.stAxisStatus.fActPosition - rActCenterX ; ;
        fbSetPosition_South.Execute := TRUE;
END_IF


//Reset
if (fbSetPosition_TOP.Done ) THEN
    fbSetPosition_TOP.Execute := FALSE;
END_IF
if (fbSetPosition_Bottom.Done ) THEN
    fbSetPosition_Bottom.Execute := FALSE;
END_IF
if (fbSetPosition_North.Done ) THEN
    fbSetPosition_North.Execute := FALSE;
END_IF
if (fbSetPosition_South.Done ) THEN
    fbSetPosition_South.Execute := FALSE;
END_IF

// Set Encoder Position
//Clear position lag error
stSetPositionOptions.ClearPositionLag := TRUE;
fbSetPosition_TOP(
    Axis:=  stTopBlade.Axis ,
    Execute:= ,
    Position:= 0 ,
    Mode:= FALSE,
    Options:= stSetPositionOptions,
    Done=> ,
    Busy=> ,
    Error=> ,
    ErrorID=> );
fbSetPosition_Bottom(
    Axis:= stBottomBlade.Axis ,
    Execute:= ,
    Position:= 0 ,
    Mode:= FALSE,
    Options:= stSetPositionOptions,
    Done=> ,
    Busy=> ,
    Error=> ,
    ErrorID=> );
fbSetPosition_North(
    Axis:= stNorthBlade.Axis ,
    Execute:= ,
    Position:= 0 ,
    Mode:= FALSE,
    Options:= stSetPositionOptions,
    Done=> ,
    Busy=> ,
    Error=> ,
    ErrorID=> );
fbSetPosition_South(
    Axis:= stSouthBlade.Axis ,
    Execute:= ,
    Position:= 0 ,
    Mode:= FALSE,
    Options:= stSetPositionOptions,
    Done=> ,
    Busy=> ,
    Error=> ,
    ErrorID=> );

    *)
END_ACTION

METHOD M_CheckPMPS : BOOL
VAR_INPUT
     index: int;
END_VAR

IF(rActApertureSizeX < (PMPS_GVL.stCurrentBeamParameters.astApertures[index].Width))
    OR (rActApertureSizeY < (PMPS_GVL.stCurrentBeamParameters.astApertures[index].Height)) THEN
        FFO.i_xOK := FALSE;
    ELSE
        FFO.i_xOK := TRUE;
END_IF

(*FAST FAULT*)
FFO(i_xOK := ,
    i_xReset := ,
    i_xAutoReset :=TRUE,
    io_fbFFHWO := this^.io_fbFFHWO);
END_METHOD

METHOD M_HomeBlade : BOOL
VAR_IN_OUT
      stBlade: DUT_MotionStage;
END_VAR
VAR
    fPosBlade: LREAL;
    HomeState: E_HomeState;
    rHomingDistance: REAL:=0.2;
    rHomingVelocity: REAL:=0.1;
    Axis: AXIS_REF;
    fbSetPosition: MC_SetPosition;
    fbWriteParameter: MC_WriteBoolParameter;
END_VAR


CASE HomeState OF
    H_READY:
        fbWriteParameter.Execute := FALSE;
        IF (bHome) THEN
            HomeState := H_INIT;
            bHomeReady := FALSE;
        END_IF


    H_INIT:
    HomeState:=H_RESET_LL;


    H_RESET_LL:
        // disable soft limits in order to be able to move the drive
        fbWriteParameter.ParameterNumber := MC_AxisParameter.EnableLimitNeg;
        fbWriteParameter.Value := FALSE;
        fbWriteParameter.Execute := TRUE;
        if (fbWriteParameter.Done) THEN
            fbWriteParameter.Execute := FALSE;
            HomeState:= H_RESET_HL;
        END_IF

    H_RESET_HL:
        // disable soft limits in order to be able to move the drive
        fbWriteParameter.ParameterNumber := MC_AxisParameter.EnableLimitPos;
        fbWriteParameter.Value := FALSE;
        fbWriteParameter.Execute := TRUE;
        if (fbWriteParameter.Done) THEN
            fbWriteParameter.Execute := FALSE;
            HomeState:= H_ENABLE;
        END_IF

    H_ENABLE:
        // Make Sure there are no errors
        IF stBlade.bError THEN
            HomeState := H_ERROR;
            ELSE
             stBlade.fPosition := stBlade.fPosition - rHomingDistance;
             HomeState:= H_MOVING;
        END_IF



    H_MOVING:
        stBlade.bExecute :=TRUE;
        IF stBlade.bBusy  THEN
            (* axis is executing job but is not yet finished *)
            stBlade.bExecute:= FALSE;
            (* leave this state and buffer a second command *)
            HomeState := H_KEEP_MOVING;
        ElSIF stBlade.bDone THEN
            stBlade.bExecute:= FALSE;
            stBlade.fPosition := stBlade.fPosition - rHomingDistance;
            HomeState := H_KEEP_MOVING;
        ELSIF stBlade.bError THEN
            stBlade.bExecute:= FALSE;
            HomeState := H_CHECK;
        END_IF

    H_KEEP_MOVING:
        IF stBlade.bError THEN
            HomeState := H_CHECK;
        END_IF
        IF  stBlade.bDone THEN
            HomeState := H_MOVING;
            stBlade.fPosition := stBlade.fPosition + rHomingDistance;
            stBlade.bExecute  := TRUE;
        END_IF

    H_CHECK:
        //Check the mpositive limit switch is reached or erro losing positive limit
        IF (stBlade.bError) AND NOT (stBlade.bLimitForwardEnable) THEN
            HomeState := H_RESET;
            stBlade.bReset := TRUE;
        ELSE
            HomeState := H_ERROR;
        END_IF

    H_RESET:
        IF NOT(stBlade.bError) THEN
            HomeState := H_SET_POS;
        END_IF

    H_SET_POS:
     // Set Current Position
        fbSetPosition.Position := 0;
        fbSetPosition.Execute := TRUE;
        IF ( fbSetPosition.Done ) THEN
            fbSetPosition.Execute := FALSE;
            HomeState:= H_WRITE_LL;
        ELSIF (fbSetPosition.Error) THEN
            HomeState := H_ERROR;
        END_IF


    H_WRITE_LL:
    // Re Enable the Soft limits
        fbWriteParameter.ParameterNumber := MC_AxisParameter.AxisEnMinSoftPosLimit;//AxisEnMaxSoftPosLimit;// .AxisEnMinSoftPosLimit;
        fbWriteParameter.Value := TRUE;
        fbWriteParameter.Execute := TRUE;
        if (fbWriteParameter.Done) THEN
            fbWriteParameter.Execute := FALSE;
            HomeState:= H_WRITE_HL;
        END_IF

    H_WRITE_HL:
    // Re Enable the Soft limits
        fbWriteParameter.ParameterNumber := MC_AxisParameter.AxisEnMaxSoftPosLimit;
        fbWriteParameter.Value := TRUE;
        fbWriteParameter.Execute := TRUE;
        if (fbWriteParameter.Done) THEN
            fbWriteParameter.Execute := FALSE;
            HomeState:= H_DONE;
        END_IF


    H_ERROR:
        //What to do?  User reset through epics??
        IF NOT (stBlade.bError) (*AND (bHome)*) THEN
            HomeState := H_INIT;
        END_IF

    H_DONE:
        HomeState := H_INIT;
        bHomeReady := TRUE;

END_CASE



// Set Encoder Position
fbSetPosition(
    Axis:= stBlade.Axis ,
    Execute:= ,
    Position:= 0 ,
    Mode:= FALSE, //Absolute
    Options:= ,
    Done=> ,
    Busy=> ,
    Error=> ,
    ErrorID=> );

// Write Parameters
fbWriteParameter(
    Axis:= stBlade.Axis ,
    Execute:= ,
    ParameterNumber:= ,
    Value:= ,
    Done=> ,
    Busy=> ,
    Error=> ,
    ErrorID=> );

If ( fbWriteParameter.Error) OR (fbSetPosition.Error) THEN
    HomeState:= H_ERROR;
END_IF
END_METHOD

METHOD M_UpdatePMPS : BOOL
VAR_INPUT
    index: int;
END_VAR
//Keep updating the status of the apertures PMPS
This^.AptArrayStatus.Height := This^.rActApertureSizeY;
This^.AptArrayStatus.Width := This^.rActApertureSizeX;
This^.AptArrayStatus.xOK := NOT (This^.stTopBlade.bError) AND NOT (This^.stBottomBlade.bError)
                                 AND NOT (This^.stNorthBlade.bError) AND NOT (This^.stNorthBlade.bError);

//Evaluate that the current center on the X and the y direction didn't exceed limits
//Fast fault when it does.
IF(rActCenterX > (PMPS_GVL.stCurrentBeamParameters.astApertures[index].Width/2))
    OR (rActCenterY > (PMPS_GVL.stCurrentBeamParameters.astApertures[index].Height/2)) THEN
        FFO.i_xOK := FALSE;
    ELSE
        FFO.i_xOK := TRUE;
END_IF

//Evaluate that the requested gaps on the X and the y direction is not larger than the current gap
// narrow  the gap if the requested is larger
IF(bTest) THEN
    IF (This^.rActApertureSizeX > AptArrayReq.Width) THEN
        rReqApertureSizeX := AptArrayReq.Width;
    END_IF
    IF (This^.rActApertureSizeY > AptArrayReq.Height) THEN
         rReqApertureSizeY := AptArrayReq.Height;
    END_IF
END_IF


(*FAST FAULT*)
FFO(i_xOK := ,
    i_xReset := ,
    i_xAutoReset :=TRUE,
    io_fbFFHWO := io_fbFFHWO);
END_METHOD

END_FUNCTION_BLOCK

// ---- POUs/PRG_ST4K4_TMO_TERM.TcPOU
PROGRAM PRG_ST4K4_TMO_TERM
VAR
    {attribute 'pytmc' := 'pv: ST4K4:TMO_TERM'}
    {attribute 'TcLinkTo' := 	'.i_xInsertedLS	:=	TIIB[ST4K4-TERM (EP2338-0001)]^Channel 4^Input;
                                 .i_xRetractedLS:=	TIIB[ST4K4-TERM (EP2338-0001)]^Channel 3^Input;
                                 .q_xRetract_DO	:=	TIIB[ST4K4-TERM (EP2338-0001)]^Channel 9^Output
    '}
    ST4K4: FB_MotionPneumaticActuator;
    ibPMPS_OK : BOOL;
    {attribute 'pytmc' :='pv: ST4K4:TMO_TERM'}
    {attribute 'TcLinkTo' := '.iRaw := TIIB[EP3174-FWM-E2]^AI Standard Channel 1^Value'}
    fbFlowMeter: FB_FDQ_FlowMeter;
END_VAR

ST4K4(
    ibInsertOK:= TRUE,
    ibRetractOK:= TRUE,
    ibPMPS_OK:= ibPMPS_OK,
    ibSingleCntrl:= TRUE ,
    ibCntrlHold:= TRUE,
    ibOverrideInterlock:= ,
    i_xReset:= ,
    i_xAutoReset := TRUE,
    stPneumaticActuator=> ,
    xMPS_OK=>  ,
    io_fbFFHWO:= fbFastFaultOutput2  ); // Do Stoppers send MPS FAULT?

// For PMPS Veto
GVL_PMPS.PMPS_ST4K4_IN := ST4K4.i_xInsertedLS;
GVL_PMPS.PMPS_ST4K4_OUT := ST4K4.i_xRetractedLS;

fbFlowMeter();

END_PROGRAM

// ---- POUs/PRG_PC5K4.TcPOU
PROGRAM PRG_PC5K4
VAR
    {attribute 'pytmc' :='pv: PC5K4'}
    {attribute 'TcLinkTo' := '.iRaw := TIIB[EP3174-FWM-E2]^AI Standard Channel 1^Value'}
    fbFlowMeter: FB_FDQ_FlowMeter;
END_VAR

fbFlowMeter();

END_PROGRAM

// ---- POUs/PRG_TM1K4.TcPOU
PROGRAM PRG_TM1K4
VAR
    {attribute 'pytmc' := '
        pv: TM1K4:ATM
        io: io
    '}
    {attribute 'TcLinkTo' := '.fbTempSensor1.bError := TIIB[TM1K4-EL3314-E5]^TC Inputs Channel 1^Status^Error;
                              .fbTempSensor1.bUnderrange := TIIB[TM1K4-EL3314-E5]^TC Inputs Channel 1^Status^Underrange;
                              .fbTempSensor1.bOverrange := TIIB[TM1K4-EL3314-E5]^TC Inputs Channel 1^Status^Overrange;
                              .fbTempSensor1.iRaw := TIIB[TM1K4-EL3314-E5]^TC Inputs Channel 1^Value;
                              .fbFlowMeter.iRaw := TIIB[IM5K4-EL3052-E5]^AI Standard Channel 1^Value'} // same cooling loop as IM5K4
    fbTM1K4: FB_TM1K4;

    bInit: BOOL;
END_VAR


IF NOT bInit THEN
    fbTM1K4.stOut.fPosition := -2.558;
    fbTM1K4.stOut.fVelocity := 1;
    fbTM1K4.stOut.sName := 'OUT';
    fbTM1K4.stOut.bUseRawCounts := FALSE;
    fbTM1K4.stOut.bValid := TRUE;
    fbTM1K4.stOut.bMoveOK := TRUE;
    fbTM1K4.stOut.stPMPS.sPmpsState := 'TM1K4:ATM-OUT';

    fbTM1K4.stTarget1a.fPosition := -15.316;
    fbTM1K4.stTarget1a.fVelocity := 1;
    fbTM1K4.stTarget1a.sName := 'clear_YAG';
    fbTM1K4.stTarget1a.bUseRawCounts := FALSE;
    fbTM1K4.stTarget1a.bValid := TRUE;
    fbTM1K4.stTarget1a.bMoveOK := TRUE;
    fbTM1K4.stTarget1a.stPMPS.sPmpsState := 'TM1K4:ATM-TARGET1a';

    fbTM1K4.stTarget1b.fPosition := -20.2167; // data is changed on 3-7-2025 due to last TMO MRCO shift
    fbTM1K4.stTarget1b.fVelocity := 1;
    fbTM1K4.stTarget1b.sName := 'GaAs_1';
    fbTM1K4.stTarget1b.bUseRawCounts := FALSE;
    fbTM1K4.stTarget1b.bValid := TRUE;
    fbTM1K4.stTarget1b.bMoveOK := TRUE;
    fbTM1K4.stTarget1b.stPMPS.sPmpsState := 'TM1K4:ATM-TARGET1b';

    fbTM1K4.stTarget2a.fPosition := -32;
    fbTM1K4.stTarget2a.fVelocity := 1;
    fbTM1K4.stTarget2a.sName := 'SiN';
    fbTM1K4.stTarget2a.bUseRawCounts := FALSE;
    fbTM1K4.stTarget2a.bValid := TRUE;
    fbTM1K4.stTarget2a.bMoveOK := TRUE;
    fbTM1K4.stTarget2a.stPMPS.sPmpsState := 'TM1K4:ATM-TARGET2a';


    fbTM1K4.stTarget2b.fPosition := -41.755;
    fbTM1K4.stTarget2b.fVelocity := 1;
    fbTM1K4.stTarget2b.sName := 'GaAs_2';
    fbTM1K4.stTarget2b.bUseRawCounts := FALSE;
    fbTM1K4.stTarget2b.bValid := TRUE;
    fbTM1K4.stTarget2b.bMoveOK := TRUE;
    fbTM1K4.stTarget2b.stPMPS.sPmpsState := 'TM1K4:ATM-TARGET2b';

    fbTM1K4.stTarget3a.fPosition := -52.318;
    fbTM1K4.stTarget3a.fVelocity := 1;
    fbTM1K4.stTarget3a.sName := 'AF_target';
    fbTM1K4.stTarget3a.bUseRawCounts := FALSE;
    fbTM1K4.stTarget3a.bValid := TRUE;
    fbTM1K4.stTarget3a.bMoveOK := TRUE;
    fbTM1K4.stTarget3a.stPMPS.sPmpsState := 'TM1K4:ATM-TARGET3a';

    fbTM1K4.stTarget3b.fPosition := -63.398;
    fbTM1K4.stTarget3b.fVelocity := 1;
    fbTM1K4.stTarget3b.sName := 'GaAs_3';
    fbTM1K4.stTarget3b.bUseRawCounts := FALSE;
    fbTM1K4.stTarget3b.bValid := TRUE;
    fbTM1K4.stTarget3b.bMoveOK := TRUE;
    fbTM1K4.stTarget3b.stPMPS.sPmpsState := 'TM1K4:ATM-TARGET3b';

    fbTM1K4.stTarget4.fPosition := -81.057;
    fbTM1K4.stTarget4.fVelocity := 1;
    fbTM1K4.stTarget4.sName := 'YAG';
    fbTM1K4.stTarget4.bUseRawCounts := FALSE;
    fbTM1K4.stTarget4.bValid := TRUE;
    fbTM1K4.stTarget4.bMoveOK := TRUE;
    fbTM1K4.stTarget4.stPMPS.sPmpsState := 'TM1K4:ATM-YAG';

    fbTM1K4.stTarget5.fPosition := -102.268;
    fbTM1K4.stTarget5.fVelocity := 1;
    fbTM1K4.stTarget5.sName := 'DIODE';
    fbTM1K4.stTarget5.bUseRawCounts := FALSE;
    fbTM1K4.stTarget5.bValid := TRUE;
    fbTM1K4.stTarget5.bMoveOK := TRUE;
    fbTM1K4.stTarget5.stPMPS.sPmpsState := 'TM1K4:ATM-DIODE';

    bInit := TRUE;
END_IF

fbTM1K4(
    fbArbiter := fbArbiter,
    fbFFHWO := fbFastFaultOutput1,
    stYStage := Main.M21,
    stXStage := Main.M22,
    sDeviceName := 'TM1K4:ATM',
    sTransitionKey := 'TM1K4:ATM-TRANSITION',
    bEnableMotion := TRUE,
    bEnableBeamParams := TRUE,
    bEnablePositionLimits := TRUE,
);

END_PROGRAM

// ---- POUs/TM1K4/FB_TM1K4.TcPOU
FUNCTION_BLOCK FB_TM1K4
(*
    Adapted from FB_ATM to:
    - Change stTarget1..stTarget5 to stTarget1a, stTarget1b, stTarget2b, stTarget3a, stTarget3b, stTarget4, stTarget5 to the inputs
    - Change the arrStates.array pragma from 1..6 to 1..9 (out and 8 in states, up from 5) // 11-08-24
    - Swap out FB_ATM_States for FB_TM1K4_States
*)
VAR_IN_OUT
    // Y motor (state select).
    stYStage: ST_MotionStage;
    // X motor (align target to beam).
    stXStage: ST_MotionStage;
    // The fast fault output to fault to.
    fbFFHWO: FB_HardwareFFOutput;
    // The arbiter to request beam conditions from.
    fbArbiter: FB_Arbiter;
END_VAR
VAR_INPUT
    stOut: ST_PositionState;
    stTarget1a: ST_PositionState;
    stTarget1b: ST_PositionState;
    stTarget2a: ST_PositionState;
    stTarget2b: ST_PositionState;
    stTarget3a: ST_PositionState;
    stTarget3b: ST_PositionState;
    stTarget4: ST_PositionState;    // target 4 is Yag
    stTarget5: ST_PositionState;    //target 5 is Diode
    // Set this to a non-unknown value to request a new move.
    {attribute 'pytmc' := '
        pv: MMS:STATE:SET
        io: io
    '}
    eEnumSet: ENUM_TM1K4_States;
    // Set this to TRUE to enable input state moves, or FALSE to disable them.
    bEnableMotion: BOOL;
    // Set this to TRUE to enable beam parameter checks, or FALSE to disable them.
    bEnableBeamParams: BOOL;
    // Set this to TRUE to enable position limit checks, or FALSE to disable them.
    bEnablePositionLimits: BOOL;
    // The name of the device for use in the PMPS DB lookup and diagnostic screens.
    sDeviceName: STRING;
    // The name of the transition state in the PMPS database.
    sTransitionKey: STRING;
    // Set this to TRUE to re-read the loaded database immediately (useful for debug).
    bReadDBNow: BOOL;
END_VAR
VAR_OUTPUT
    // The current position state as an enum.
    {attribute 'pytmc' := '
        pv: MMS:STATE:GET
        io: i
    '}
    eEnumGet: ENUM_TM1K4_States;
    // The PMPS database lookup associated with the current position state.
    stDbStateParams: ST_DbStateParams;
END_VAR
VAR
    bInit: BOOL;

    fbYStage: FB_MotionStage;
    fbXStage: FB_MotionStage;

    fbStateDefaults: FB_PositionState_Defaults;

    {attribute 'pytmc' := '
        pv: MMS
        astPositionState.array: 1..9
    '}
    fbStates: FB_PositionStatePMPS1D;
    astPositionState: ARRAY[1..GeneralConstants.MAX_STATES] OF ST_PositionState;
    fbArrCheckWrite: FB_CheckPositionStateWrite;

    {attribute 'pytmc' := 'pv: STC:01'}
    fbTempSensor1: FB_CC_TempSensor;

    {attribute 'pytmc' :='pv: FWM'}
    fbFlowMeter: FB_AnalogInput := (iTermBits:=15, fTermMax:=60, fTermMin:=0);
END_VAR
VAR CONSTANT
    // State defaults if not provided
    fDelta: LREAL := 2;
    fAccel: LREAL := 200;
    fOutDecel: LREAL := 25;
END_VAR

IF NOT bInit THEN
    bInit := TRUE;

    stYStage.nEnableMode := ENUM_StageEnableMode.DURING_MOTION;
    stXStage.nEnableMode := ENUM_StageEnableMode.DURING_MOTION;

    // Partial backcompat, this used to set fVelocity too but this should be set per install
    fbStateDefaults(stPositionState:=stOut, sNameDefault:='OUT', fDeltaDefault:=fDelta, fAccelDefault:=fAccel, fDecelDefault:=fOutDecel);
    fbStateDefaults(stPositionState:=stTarget1a, sNameDefault:='TARGET1a', fDeltaDefault:=fDelta, fAccelDefault:=fAccel, fDecelDefault:=fAccel);
    fbStateDefaults(stPositionState:=stTarget1b, sNameDefault:='TARGET1b', fDeltaDefault:=fDelta, fAccelDefault:=fAccel, fDecelDefault:=fAccel);
    fbStateDefaults(stPositionState:=stTarget2a, sNameDefault:='TARGET2a', fDeltaDefault:=fDelta, fAccelDefault:=fAccel, fDecelDefault:=fAccel);
    fbStateDefaults(stPositionState:=stTarget2b, sNameDefault:='TARGET2b', fDeltaDefault:=fDelta, fAccelDefault:=fAccel, fDecelDefault:=fAccel);
    fbStateDefaults(stPositionState:=stTarget3a, sNameDefault:='TARGET3a', fDeltaDefault:=fDelta, fAccelDefault:=fAccel, fDecelDefault:=fAccel);
    fbStateDefaults(stPositionState:=stTarget3b, sNameDefault:='TARGET3b', fDeltaDefault:=fDelta, fAccelDefault:=fAccel, fDecelDefault:=fAccel);
    fbStateDefaults(stPositionState:=stTarget4, sNameDefault:='YAG', fDeltaDefault:=fDelta, fAccelDefault:=fAccel, fDecelDefault:=fAccel);
    fbStateDefaults(stPositionState:=stTarget5, sNameDefault:='DIODE', fDeltaDefault:=fDelta, fAccelDefault:=fAccel, fDecelDefault:=fAccel);
END_IF

stYStage.bHardwareEnable := TRUE;
stYStage.bPowerSelf := FALSE;

stXStage.bLimitForwardEnable := TRUE;
stXStage.bLimitBackwardEnable := TRUE;
stXStage.bHardwareEnable := TRUE;
stXStage.bPowerSelf := TRUE;

fbYStage(stMotionStage:=stYStage);
fbXStage(stMotionStage:=stXStage);

// We need to update from PLC or from EPICS, but not both
fbArrCheckWrite(
    astPositionState:=astPositionState,
    bCheck:=TRUE,
    bSave:=FALSE,
);
IF NOT fbArrCheckWrite.bHadWrite THEN
    astPositionState[ENUM_TM1K4_States.OUT] := stOut;
    astPositionState[ENUM_TM1K4_States.TARGET1a] := stTarget1a;
    astPositionState[ENUM_TM1K4_States.TARGET1b] := stTarget1b;
    astPositionState[ENUM_TM1K4_States.TARGET2a] := stTarget2a;
    astPositionState[ENUM_TM1K4_States.TARGET2b] := stTarget2b;
    astPositionState[ENUM_TM1K4_States.TARGET3a] := stTarget3a;
    astPositionState[ENUM_TM1K4_States.TARGET3b] := stTarget3b;
    astPositionState[ENUM_TM1K4_States.YAG] := stTarget4;
    astPositionState[ENUM_TM1K4_States.DIODE] := stTarget5;
END_IF

fbStates(
    stMotionStage:=stYStage,
    astPositionState:=astPositionState,
    eEnumSet:=eEnumSet,
    eEnumGet:=eEnumGet,
    fbFFHWO:=fbFFHWO,
    fbArbiter:=fbArbiter,
    bEnableMotion:=bEnableMotion,
    bEnableBeamParams:=bEnableBeamParams,
    bEnablePositionLimits:=bEnablePositionLimits,
    sDeviceName:=sDeviceName,
    sTransitionKey:=sTransitionKey,
    bReadDBNow:=bReadDBNow,
    stDbStateParams=>stDbStateParams,
);

fbArrCheckWrite(
    astPositionState:=astPositionState,
    bCheck:=FALSE,
    bSave:=TRUE,
);

stOut := astPositionState[ENUM_TM1K4_States.OUT];
stTarget1a := astPositionState[ENUM_TM1K4_States.TARGET1a];
stTarget1b := astPositionState[ENUM_TM1K4_States.TARGET1b];
stTarget2a := astPositionState[ENUM_TM1K4_States.TARGET2a];
stTarget2b := astPositionState[ENUM_TM1K4_States.TARGET2b];
stTarget3a := astPositionState[ENUM_TM1K4_States.TARGET3a];
stTarget3b := astPositionState[ENUM_TM1K4_States.TARGET3b];
stTarget4 := astPositionState[ENUM_TM1K4_States.YAG];
stTarget5 := astPositionState[ENUM_TM1K4_States.DIODE];

fbTempSensor1(
    fFaultThreshold:=fbStates.stDbStateParams.stReactiveParams.nTempSP,
    bVeto:=eEnumGet = ENUM_TM1K4_States.OUT,
    sDevName:=sDeviceName,
    io_fbFFHWO:=fbFFHWO,
);
fbFlowMeter();

END_FUNCTION_BLOCK

// ---- POUs/PRG_TM2K4.TcPOU
PROGRAM PRG_TM2K4
VAR
    {attribute 'pytmc' := '
        pv: TM2K4:ATM
        io: io
    '}
    {attribute 'TcLinkTo' := '.fbTempSensor1.bError := TIIB[TM2K4-EL3314-E5]^TC Inputs Channel 1^Status^Error;
                              .fbTempSensor1.bUnderrange := TIIB[TM2K4-EL3314-E5]^TC Inputs Channel 1^Status^Underrange;
                              .fbTempSensor1.bOverrange := TIIB[TM2K4-EL3314-E5]^TC Inputs Channel 1^Status^Overrange;
                              .fbTempSensor1.iRaw := TIIB[TM2K4-EL3314-E5]^TC Inputs Channel 1^Value;
                              .fbFlowMeter.iRaw := TIIB[IM6K4-EL3052-E5]^AI Standard Channel 1^Value'} // same as IM6K4
    fbTM2K4: FB_TM2K4;

    bInit: BOOL;
END_VAR



IF NOT bInit THEN
    fbTM2K4.stOut.fPosition := -1.558;
    fbTM2K4.stOut.fVelocity := 1;
    fbTM2K4.stOut.bUseRawCounts := FALSE;
    fbTM2K4.stOut.bValid := TRUE;
    fbTM2K4.stOut.sName := 'OUT';
    fbTM2K4.stOut.bMoveOK := TRUE;
    fbTM2K4.stOut.stPMPS.sPmpsState := 'TM2K4:ATM-OUT';

    fbTM2K4.stTarget1a.fPosition := -10.5;
    fbTM2K4.stTarget1a.fVelocity := 1;
    fbTM2K4.stTarget1a.bUseRawCounts := FALSE;
    fbTM2K4.stTarget1a.bValid := TRUE;
    fbTM2K4.stTarget1a.sName := 'InGaAs_1';
    fbTM2K4.stTarget1a.bMoveOK := TRUE;
   fbTM2K4.stTarget1a.stPMPS.sPmpsState := 'TM2K4:ATM-TARGET1a';

    fbTM2K4.stTarget1b.fPosition := -16.5;
    fbTM2K4.stTarget1b.fVelocity := 1;
    fbTM2K4.stTarget1b.bUseRawCounts := FALSE;
    fbTM2K4.stTarget1b.bValid := TRUE;
    fbTM2K4.stTarget1b.sName := 'InGaAs_2';
    fbTM2K4.stTarget1b.bMoveOK := TRUE;
   fbTM2K4.stTarget1b.stPMPS.sPmpsState := 'TM2K4:ATM-TARGET1b';

    fbTM2K4.stTarget2a.fPosition := -31.5;
    fbTM2K4.stTarget2a.fVelocity := 1;
    fbTM2K4.stTarget2a.bUseRawCounts := FALSE;
    fbTM2K4.stTarget2a.bValid := TRUE;
    fbTM2K4.stTarget2a.sName := 'GaAs_1';
    fbTM2K4.stTarget2a.bMoveOK := TRUE;
    fbTM2K4.stTarget2a.stPMPS.sPmpsState := 'TM2K4:ATM-TARGET2a';

    fbTM2K4.stTarget2b.fPosition := -38.5;
    fbTM2K4.stTarget2b.fVelocity := 1;
    fbTM2K4.stTarget2b.bUseRawCounts := FALSE;
    fbTM2K4.stTarget2b.bValid := TRUE;
    fbTM2K4.stTarget2b.sName := 'GaAs_2';
    fbTM2K4.stTarget2b.bMoveOK := TRUE;
    fbTM2K4.stTarget2b.stPMPS.sPmpsState := 'TM2K4:ATM-TARGET2b';


    fbTM2K4.stTarget3a.fPosition := -53.5;
    fbTM2K4.stTarget3a.fVelocity := 1;
    fbTM2K4.stTarget3a.bUseRawCounts := FALSE;
    fbTM2K4.stTarget3a.bValid := TRUE;
    fbTM2K4.stTarget3a.sName := 'gITO';
    fbTM2K4.stTarget3a.bMoveOK := TRUE;
    fbTM2K4.stTarget3a.stPMPS.sPmpsState := 'TM2K4:ATM-TARGET3a';

    fbTM2K4.stTarget3b.fPosition := -57.5;
    fbTM2K4.stTarget3b.fVelocity := 1;
    fbTM2K4.stTarget3b.bUseRawCounts := FALSE;
    fbTM2K4.stTarget3b.bValid := TRUE;
    fbTM2K4.stTarget3b.sName := 'AF_target';
    fbTM2K4.stTarget3b.bMoveOK := TRUE;
    fbTM2K4.stTarget3b.stPMPS.sPmpsState := 'TM2K4:ATM-TARGET3b';

    fbTM2K4.stTarget4.fPosition := -77.5;
    fbTM2K4.stTarget4.fVelocity := 1;
    fbTM2K4.stTarget4.bUseRawCounts := FALSE;
    fbTM2K4.stTarget4.bValid := TRUE;
    fbTM2K4.stTarget4.bMoveOK := TRUE;
    fbTM2K4.stTarget4.sName := 'YAG';
    fbTM2K4.stTarget4.stPMPS.sPmpsState := 'TM2K4:ATM-YAG';

    fbTM2K4.stTarget5.fPosition := -102.5;
    fbTM2K4.stTarget5.fVelocity := 1;
    fbTM2K4.stTarget5.bUseRawCounts := FALSE;
    fbTM2K4.stTarget5.bValid := TRUE;
    fbTM2K4.stTarget5.sName := 'DIODE';
    fbTM2K4.stTarget5.bMoveOK := TRUE;
    fbTM2K4.stTarget5.stPMPS.sPmpsState := 'TM2K4:ATM-DIODE';

    bInit := TRUE;
END_IF


fbTM2K4(
    fbArbiter := fbArbiter2,
    fbFFHWO := fbFastFaultOutput2,
    stYStage := Main.M30,
    stXStage := Main.M31,
    sDeviceName := 'TM2K4:ATM',
    sTransitionKey := 'TM2K4:ATM-TRANSITION',
    bEnableMotion := TRUE,
    bEnableBeamParams := TRUE,
    bEnablePositionLimits := TRUE,
);

END_PROGRAM

// ---- POUs/TM2K4/FB_TM2K4.TcPOU
FUNCTION_BLOCK FB_TM2K4
(*
    Adapted from FB_ATM to:
    - Change stTarget1..stTarget5 to stTarget1a, stTarget1b, stTarget2b, stTarget3a, stTarget3b, stTarget4, stTarget5 to the inputs
    - Change the arrStates.array pragma from 1..6 to 1..9 (out and 8 in states, up from 5)
    - Swap out FB_ATM_States for FB_TM2K4_States //04-2025
*)
VAR_IN_OUT
    // Y motor (state select).
    stYStage: ST_MotionStage;
    // X motor (align target to beam).
    stXStage: ST_MotionStage;
    // The fast fault output to fault to.
    fbFFHWO: FB_HardwareFFOutput;
    // The arbiter to request beam conditions from.
    fbArbiter: FB_Arbiter;
END_VAR
VAR_INPUT
    stOut: ST_PositionState;
    stTarget1a: ST_PositionState;
    stTarget1b: ST_PositionState;
    stTarget2a: ST_PositionState;
    stTarget2b: ST_PositionState;
    stTarget3a: ST_PositionState;
    stTarget3b: ST_PositionState;
    stTarget4: ST_PositionState;    // target 4 is Yag
    stTarget5: ST_PositionState;    //target 5 is Diode
    // Set this to a non-unknown value to request a new move.
    {attribute 'pytmc' := '
        pv: MMS:STATE:SET
        io: io
    '}
    eEnumSet: ENUM_TM2K4_States;
    // Set this to TRUE to enable input state moves, or FALSE to disable them.
    bEnableMotion: BOOL;
    // Set this to TRUE to enable beam parameter checks, or FALSE to disable them.
    bEnableBeamParams: BOOL;
    // Set this to TRUE to enable position limit checks, or FALSE to disable them.
    bEnablePositionLimits: BOOL;
    // The name of the device for use in the PMPS DB lookup and diagnostic screens.
    sDeviceName: STRING;
    // The name of the transition state in the PMPS database.
    sTransitionKey: STRING;
    // Set this to TRUE to re-read the loaded database immediately (useful for debug).
    bReadDBNow: BOOL;
END_VAR
VAR_OUTPUT
    // The current position state as an enum.
    {attribute 'pytmc' := '
        pv: MMS:STATE:GET
        io: i
    '}
    eEnumGet: ENUM_TM2K4_States;
    // The PMPS database lookup associated with the current position state.
    stDbStateParams: ST_DbStateParams;
END_VAR
VAR
    bInit: BOOL;

    fbYStage: FB_MotionStage;
    fbXStage: FB_MotionStage;

    fbStateDefaults: FB_PositionState_Defaults;

    {attribute 'pytmc' := '
        pv: MMS
        astPositionState.array: 1..9
    '}
    fbStates: FB_PositionStatePMPS1D;
    astPositionState: ARRAY[1..GeneralConstants.MAX_STATES] OF ST_PositionState;
    fbArrCheckWrite: FB_CheckPositionStateWrite;

    {attribute 'pytmc' := 'pv: STC:01'}
    fbTempSensor1: FB_CC_TempSensor;

    {attribute 'pytmc' :='pv: FWM'}
    fbFlowMeter: FB_AnalogInput := (iTermBits:=15, fTermMax:=60, fTermMin:=0);
END_VAR
VAR CONSTANT
    // State defaults if not provided
    fDelta: LREAL := 2;
    fAccel: LREAL := 200;
    fOutDecel: LREAL := 25;
END_VAR

IF NOT bInit THEN
    bInit := TRUE;

    stYStage.nEnableMode := ENUM_StageEnableMode.DURING_MOTION;
    stXStage.nEnableMode := ENUM_StageEnableMode.DURING_MOTION;

    // Partial backcompat, this used to set fVelocity too but this should be set per install
    fbStateDefaults(stPositionState:=stOut, sNameDefault:='OUT', fDeltaDefault:=fDelta, fAccelDefault:=fAccel, fDecelDefault:=fOutDecel);
    fbStateDefaults(stPositionState:=stTarget1a, sNameDefault:='TARGET1a', fDeltaDefault:=fDelta, fAccelDefault:=fAccel, fDecelDefault:=fAccel);
    fbStateDefaults(stPositionState:=stTarget1b, sNameDefault:='TARGET1b', fDeltaDefault:=fDelta, fAccelDefault:=fAccel, fDecelDefault:=fAccel);
    fbStateDefaults(stPositionState:=stTarget2a, sNameDefault:='TARGET2a', fDeltaDefault:=fDelta, fAccelDefault:=fAccel, fDecelDefault:=fAccel);
    fbStateDefaults(stPositionState:=stTarget2b, sNameDefault:='TARGET2b', fDeltaDefault:=fDelta, fAccelDefault:=fAccel, fDecelDefault:=fAccel);
    fbStateDefaults(stPositionState:=stTarget3a, sNameDefault:='TARGET3a', fDeltaDefault:=fDelta, fAccelDefault:=fAccel, fDecelDefault:=fAccel);
    fbStateDefaults(stPositionState:=stTarget3b, sNameDefault:='TARGET3b', fDeltaDefault:=fDelta, fAccelDefault:=fAccel, fDecelDefault:=fAccel);
    fbStateDefaults(stPositionState:=stTarget4, sNameDefault:='YAG', fDeltaDefault:=fDelta, fAccelDefault:=fAccel, fDecelDefault:=fAccel);
    fbStateDefaults(stPositionState:=stTarget5, sNameDefault:='DIODE', fDeltaDefault:=fDelta, fAccelDefault:=fAccel, fDecelDefault:=fAccel);
END_IF

stYStage.bHardwareEnable := TRUE;
stYStage.bPowerSelf := FALSE;

